KUKA KRL program: f1_Kuka_APT201T03S01.SRC

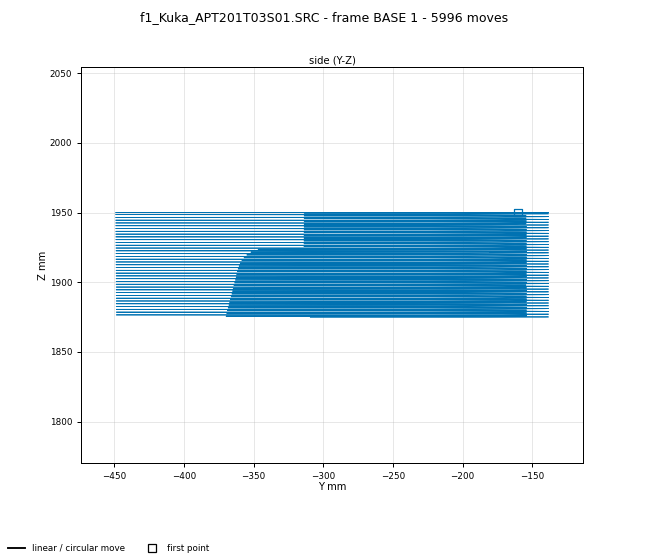
[picture p0: tool path of f1_Kuka_APT201T03S01.SRC in frame BASE 1, 5996 of 5998 moves have a stored position in this frame; points joined in program order, loops and branches not executed]
&ACCESS RVP
&REL 2
&PARAM TEMPLATE = C:\KRC\Roboter\Template\vorgabe
&PARAM EDITMASK = *
DEF f1_Kuka_APT201T03S01()


;FOLD INI;%{PE}%V3.2.0,%MKUKATPBASIS,%CINIT,%VCOMMON,%P
  ;FOLD BAS INI;%{E}%V3.2.0,%MKUKATPBASIS,%CINIT,%VINIT,%P
    GLOBAL INTERRUPT DECL 3 WHEN $STOPMESS==TRUE DO IR_STOPM ( )
    INTERRUPT ON 3
    BAS (#INITMOV,0 )
  ;ENDFOLD (BAS INI)
  ;FOLD USER INI;%{E}%V3.2.0,%MKUKATPUSER,%CINIT,%VINIT,%P
    ;Make your modifications here
  ;ENDFOLD (USER INI)
;ENDFOLD (INI)



;*** Make Initial Position Move
;FOLD PTP PPI1  Vel= 100 % PDAT1 Tool[0] Base[0];%{PE}%R 5.2.22,%MKUKATPBASIS,%CMOVE,%VPTP,%P 1:PTP, 2:PPI1, 3:, 5:100, 7:PDAT1
  $BWDSTART = FALSE
  PDAT_ACT = PPDAT1
  FDAT_ACT = FPPI1
  BAS(#PTP_PARAMS,100)
  PTP XPPI1
;ENDFOLD


;*** Auto Load the Correct TOOL and OFFSET
  ToolChange(3,1)


;*** Make Initial Position Move
;FOLD PTP PPI1  Vel= 100 % PDAT1 Tool[0] Base[0];%{PE}%R 5.2.22,%MKUKATPBASIS,%CMOVE,%VPTP,%P 1:PTP, 2:PPI1, 3:, 5:100, 7:PDAT1
  $BWDSTART = FALSE
  PDAT_ACT = PPDAT1
  FDAT_ACT = FPPI1
  BAS(#PTP_PARAMS,100)
  PTP XPPI1
;ENDFOLD

;*** Auto Load The Correct TOOL Data
  $tool=tool_data[3]

;*** Auto Load The Correct BASE Data
  $base=base_data[1]

  $ADVANCE = 5

SetRPM(6000)

MMPM(30000.0)
LIN {X 0.000,Y -160.097,Z 1950.000,A 0.000,B 0.000,C 90.000,E1 360.000} C_DIS
MMPM(15000.0)
LIN {X 0.000,Y -155.097,Z 1950.000,A 0.000,B 0.000,C 90.000,E1 360.000} C_DIS
MMPM(30000.0)
LIN {X -0.008,Y -154.165,Z 1950.000,A 0.000,B 0.000,C 90.000,E1 352.356} C_DIS
LIN {X -0.016,Y -155.912,Z 1950.000,A 0.000,B 0.000,C 90.000,E1 344.283} C_DIS
LIN {X 0.049,Y -158.612,Z 1950.000,A 0.000,B 0.000,C 90.000,E1 338.901} C_DIS
LIN {X 0.065,Y -162.189,Z 1950.000,A 0.000,B 0.000,C 90.000,E1 334.460} C_DIS
LIN {X -0.028,Y -166.034,Z 1950.000,A 0.000,B 0.000,C 90.000,E1 330.973} C_DIS
LIN {X 0.069,Y -170.880,Z 1950.000,A 0.000,B 0.000,C 90.000,E1 327.454} C_DIS
LIN {X -0.020,Y -175.155,Z 1950.000,A 0.000,B 0.000,C 90.000,E1 324.895} C_DIS
LIN {X -0.079,Y -180.105,Z 1950.000,A 0.000,B 0.000,C 90.000,E1 322.351} C_DIS
LIN {X 0.029,Y -185.957,Z 1950.000,A 0.000,B 0.000,C 90.000,E1 319.784} C_DIS
LIN {X -0.007,Y -191.568,Z 1950.000,A 0.000,B 0.000,C 90.000,E1 317.715} C_DIS
LIN {X 0.028,Y -199.262,Z 1950.000,A 0.000,B 0.000,C 90.000,E1 315.243} C_DIS
LIN {X -0.070,Y -207.846,Z 1950.000,A 0.000,B 0.000,C 90.000,E1 312.852} C_DIS
LIN {X -0.093,Y -218.894,Z 1950.000,A 0.000,B 0.000,C 90.000,E1 310.092} C_DIS
LIN {X -0.030,Y -232.809,Z 1950.000,A 0.000,B 0.000,C 90.000,E1 306.996} C_DIS
LIN {X 0.030,Y -247.857,Z 1950.000,A 0.000,B 0.000,C 90.000,E1 303.992} C_DIS
LIN {X 0.078,Y -259.781,Z 1950.000,A 0.000,B 0.000,C 90.000,E1 301.799} C_DIS
LIN {X 0.080,Y -271.838,Z 1950.000,A 0.000,B 0.000,C 90.000,E1 299.667} C_DIS
LIN {X -0.149,Y -281.753,Z 1950.000,A 0.000,B 0.000,C 90.000,E1 297.975} C_DIS
LIN {X 0.022,Y -291.348,Z 1950.000,A 0.000,B 0.000,C 90.000,E1 296.232} C_DIS
LIN {X 0.102,Y -296.741,Z 1950.000,A 0.000,B 0.000,C 90.000,E1 295.207} C_DIS
LIN {X 0.101,Y -301.534,Z 1950.000,A 0.000,B 0.000,C 90.000,E1 294.207} C_DIS
LIN {X -0.014,Y -304.343,Z 1950.000,A 0.000,B 0.000,C 90.000,E1 293.567} C_DIS
LIN {X 0.047,Y -306.751,Z 1950.000,A 0.000,B 0.000,C 90.000,E1 292.898} C_DIS
LIN {X -0.041,Y -308.757,Z 1950.000,A 0.000,B 0.000,C 90.000,E1 292.259} C_DIS
LIN {X 0.048,Y -310.413,Z 1950.000,A 0.000,B 0.000,C 90.000,E1 291.589} C_DIS
LIN {X 0.151,Y -311.750,Z 1950.000,A 0.000,B 0.000,C 90.000,E1 290.918} C_DIS
LIN {X -0.026,Y -312.741,Z 1950.000,A 0.000,B 0.000,C 90.000,E1 290.301} C_DIS
LIN {X 0.097,Y -313.399,Z 1950.000,A 0.000,B 0.000,C 90.000,E1 289.631} C_DIS
LIN {X -0.070,Y -313.739,Z 1950.000,A 0.000,B 0.000,C 90.000,E1 289.014} C_DIS
LIN {X -0.038,Y -313.728,Z 1950.000,A 0.000,B 0.000,C 90.000,E1 288.362} C_DIS
LIN {X 0.095,Y -313.339,Z 1950.000,A 0.000,B 0.000,C 90.000,E1 287.692} C_DIS
LIN {X 0.134,Y -312.501,Z 1950.000,A 0.000,B 0.000,C 90.000,E1 287.040} C_DIS
LIN {X -0.127,Y -311.193,Z 1950.000,A 0.000,B 0.000,C 90.000,E1 286.441} C_DIS
LIN {X -0.093,Y -309.374,Z 1950.000,A 0.000,B 0.000,C 90.000,E1 285.788} C_DIS
LIN {X -0.067,Y -306.893,Z 1950.000,A 0.000,B 0.000,C 90.000,E1 285.134} C_DIS
LIN {X -0.058,Y -303.660,Z 1950.000,A 0.000,B 0.000,C 90.000,E1 284.481} C_DIS
LIN {X -0.103,Y -295.919,Z 1950.000,A 0.000,B 0.000,C 90.000,E1 283.175} C_DIS
LIN {X -0.023,Y -290.732,Z 1950.000,A 0.000,B 0.000,C 90.000,E1 282.187} C_DIS
LIN {X -0.115,Y -286.366,Z 1950.000,A 0.000,B 0.000,C 90.000,E1 281.535} C_DIS
LIN {X -0.010,Y -281.038,Z 1950.000,A 0.000,B 0.000,C 90.000,E1 280.838} C_DIS
LIN {X -0.011,Y -274.872,Z 1950.000,A 0.000,B 0.000,C 90.000,E1 280.197} C_DIS
LIN {X 0.056,Y -268.439,Z 1950.000,A 0.000,B 0.000,C 90.000,E1 279.613} C_DIS
LIN {X 0.112,Y -261.807,Z 1950.000,A 0.000,B 0.000,C 90.000,E1 279.095} C_DIS
LIN {X -0.044,Y -255.112,Z 1950.000,A 0.000,B 0.000,C 90.000,E1 278.681} C_DIS
LIN {X 0.015,Y -248.167,Z 1950.000,A 0.000,B 0.000,C 90.000,E1 278.276} C_DIS
LIN {X 0.073,Y -240.768,Z 1950.000,A 0.000,B 0.000,C 90.000,E1 277.936} C_DIS
LIN {X -0.029,Y -232.686,Z 1950.000,A 0.000,B 0.000,C 90.000,E1 277.701} C_DIS
LIN {X -0.115,Y -222.350,Z 1950.000,A 0.000,B 0.000,C 90.000,E1 277.530} C_DIS
LIN {X -0.092,Y -214.660,Z 1950.000,A 0.000,B 0.000,C 90.000,E1 277.466} C_DIS
LIN {X 0.070,Y -180.206,Z 1950.000,A 0.000,B 0.000,C 90.000,E1 277.409} C_DIS
LIN {X 0.037,Y -181.028,Z 1950.000,A 0.000,B 0.000,C 90.000,E1 275.391} C_DIS
LIN {X 0.012,Y -181.579,Z 1950.000,A 0.000,B 0.000,C 90.000,E1 270.344} C_DIS
LIN {X -0.013,Y -180.904,Z 1950.000,A 0.000,B 0.000,C 90.000,E1 265.298} C_DIS
LIN {X -0.063,Y -180.241,Z 1950.000,A 0.000,B 0.000,C 90.000,E1 263.628} C_DIS
LIN {X -0.044,Y -178.728,Z 1950.000,A 0.000,B 0.000,C 90.000,E1 259.398} C_DIS
LIN {X 0.024,Y -175.777,Z 1950.000,A 0.000,B 0.000,C 90.000,E1 254.283} C_DIS
LIN {X 0.011,Y -171.961,Z 1950.000,A 0.000,B 0.000,C 90.000,E1 249.156} C_DIS
LIN {X 0.048,Y -171.355,Z 1950.000,A 0.000,B 0.000,C 90.000,E1 248.284} C_DIS
LIN {X 0.026,Y -167.605,Z 1950.000,A 0.000,B 0.000,C 90.000,E1 243.973} C_DIS
LIN {X 0.039,Y -166.250,Z 1950.000,A 0.000,B 0.000,C 90.000,E1 242.231} C_DIS
LIN {X 0.026,Y -163.005,Z 1950.000,A 0.000,B 0.000,C 90.000,E1 238.742} C_DIS
LIN {X 0.073,Y -160.927,Z 1950.000,A 0.000,B 0.000,C 90.000,E1 236.087} C_DIS
LIN {X 0.050,Y -157.689,Z 1950.000,A 0.000,B 0.000,C 90.000,E1 232.557} C_DIS
LIN {X -0.012,Y -155.727,Z 1950.000,A 0.000,B 0.000,C 90.000,E1 229.908} C_DIS
LIN {X 0.042,Y -151.987,Z 1950.000,A 0.000,B 0.000,C 90.000,E1 225.405} C_DIS
LIN {X 0.058,Y -150.231,Z 1950.000,A 0.000,B 0.000,C 90.000,E1 222.690} C_DIS
LIN {X -0.019,Y -146.992,Z 1950.000,A 0.000,B 0.000,C 90.000,E1 218.177} C_DIS
LIN {X -0.029,Y -145.577,Z 1950.000,A 0.000,B 0.000,C 90.000,E1 215.438} C_DIS
LIN {X -0.035,Y -142.967,Z 1950.000,A 0.000,B 0.000,C 90.000,E1 210.846} C_DIS
LIN {X 0.019,Y -141.593,Z 1950.000,A 0.000,B 0.000,C 90.000,E1 207.129} C_DIS
LIN {X 0.065,Y -139.421,Z 1950.000,A 0.000,B 0.000,C 90.000,E1 200.610} C_DIS
LIN {X -0.014,Y -139.148,Z 1950.000,A 0.000,B 0.000,C 90.000,E1 198.779} C_DIS
LIN {X 0.008,Y -138.346,Z 1950.000,A 0.000,B 0.000,C 90.000,E1 190.366} C_DIS
LIN {X -0.006,Y -139.487,Z 1950.000,A 0.000,B 0.000,C 90.000,E1 181.031} C_DIS
LIN {X -0.066,Y -141.091,Z 1950.000,A 0.000,B 0.000,C 90.000,E1 175.469} C_DIS
LIN {X 0.028,Y -142.469,Z 1950.000,A 0.000,B 0.000,C 90.000,E1 172.648} C_DIS
LIN {X -0.024,Y -144.713,Z 1950.000,A 0.000,B 0.000,C 90.000,E1 168.049} C_DIS
LIN {X 0.069,Y -147.314,Z 1950.000,A 0.000,B 0.000,C 90.000,E1 164.338} C_DIS
LIN {X -0.058,Y -150.634,Z 1950.000,A 0.000,B 0.000,C 90.000,E1 159.826} C_DIS
LIN {X 0.018,Y -154.111,Z 1950.000,A 0.000,B 0.000,C 90.000,E1 156.177} C_DIS
LIN {X -0.058,Y -157.536,Z 1950.000,A 0.000,B 0.000,C 90.000,E1 152.615} C_DIS
LIN {X 0.107,Y -161.773,Z 1950.000,A 0.000,B 0.000,C 90.000,E1 148.997} C_DIS
LIN {X -0.010,Y -165.966,Z 1950.000,A 0.000,B 0.000,C 90.000,E1 145.515} C_DIS
LIN {X -0.013,Y -170.959,Z 1950.000,A 0.000,B 0.000,C 90.000,E1 142.029} C_DIS
LIN {X 0.038,Y -175.828,Z 1950.000,A 0.000,B 0.000,C 90.000,E1 138.566} C_DIS
LIN {X 0.033,Y -181.435,Z 1950.000,A 0.000,B 0.000,C 90.000,E1 135.162} C_DIS
LIN {X -0.093,Y -186.940,Z 1950.000,A 0.000,B 0.000,C 90.000,E1 131.838} C_DIS
LIN {X -0.094,Y -190.052,Z 1950.000,A 0.000,B 0.000,C 90.000,E1 130.172} C_DIS
LIN {X -0.079,Y -195.827,Z 1950.000,A 0.000,B 0.000,C 90.000,E1 126.870} C_DIS
LIN {X -0.012,Y -200.659,Z 1950.000,A 0.000,B 0.000,C 90.000,E1 124.405} C_DIS
LIN {X 0.005,Y -206.543,Z 1950.000,A 0.000,B 0.000,C 90.000,E1 121.180} C_DIS
LIN {X -0.008,Y -209.835,Z 1950.000,A 0.000,B 0.000,C 90.000,E1 119.589} C_DIS
LIN {X -0.083,Y -217.193,Z 1950.000,A 0.000,B 0.000,C 90.000,E1 115.668} C_DIS
LIN {X 0.070,Y -218.819,Z 1950.000,A 0.000,B 0.000,C 90.000,E1 114.847} C_DIS
LIN {X 0.093,Y -224.206,Z 1950.000,A 0.000,B 0.000,C 90.000,E1 111.770} C_DIS
LIN {X 0.086,Y -283.482,Z 1950.000,A 0.000,B 0.000,C 90.000,E1 111.770} C_DIS
LIN {X -0.008,Y -285.142,Z 1950.000,A 0.000,B 0.000,C 90.000,E1 111.770} C_DIS
LIN {X -0.069,Y -288.414,Z 1950.000,A 0.000,B 0.000,C 90.000,E1 111.663} C_DIS
LIN {X 0.069,Y -291.624,Z 1950.000,A 0.000,B 0.000,C 90.000,E1 111.408} C_DIS
LIN {X 0.113,Y -295.303,Z 1950.000,A 0.000,B 0.000,C 90.000,E1 110.972} C_DIS
LIN {X 0.154,Y -300.812,Z 1950.000,A 0.000,B 0.000,C 90.000,E1 109.993} C_DIS
LIN {X 0.157,Y -314.505,Z 1950.000,A 0.000,B 0.000,C 90.000,E1 107.692} C_DIS
LIN {X -0.024,Y -329.600,Z 1950.000,A 0.000,B 0.000,C 90.000,E1 105.481} C_DIS
LIN {X 0.050,Y -343.764,Z 1950.000,A 0.000,B 0.000,C 90.000,E1 103.592} C_DIS
LIN {X 0.020,Y -359.097,Z 1950.000,A 0.000,B 0.000,C 90.000,E1 101.771} C_DIS
LIN {X 0.045,Y -377.683,Z 1950.000,A 0.000,B 0.000,C 90.000,E1 99.792} C_DIS
LIN {X 0.102,Y -396.651,Z 1950.000,A 0.000,B 0.000,C 90.000,E1 97.992} C_DIS
LIN {X 0.049,Y -418.788,Z 1950.000,A 0.000,B 0.000,C 90.000,E1 96.144} C_DIS
LIN {X 0.229,Y -438.507,Z 1950.000,A 0.000,B 0.000,C 90.000,E1 94.645} C_DIS
LIN {X -0.197,Y -442.974,Z 1950.000,A 0.000,B 0.000,C 90.000,E1 94.302} C_DIS
LIN {X 0.177,Y -446.090,Z 1950.000,A 0.000,B 0.000,C 90.000,E1 93.784} C_DIS
LIN {X -0.091,Y -447.256,Z 1950.000,A 0.000,B 0.000,C 90.000,E1 93.555} C_DIS
LIN {X 0.089,Y -448.110,Z 1950.000,A 0.000,B 0.000,C 90.000,E1 93.269} C_DIS
LIN {X 0.052,Y -449.023,Z 1950.000,A 0.000,B 0.000,C 90.000,E1 92.751} C_DIS
LIN {X -0.002,Y -448.993,Z 1950.000,A 0.000,B 0.000,C 90.000,E1 92.236} C_DIS
LIN {X -0.035,Y -448.019,Z 1950.000,A 0.000,B 0.000,C 90.000,E1 91.718} C_DIS
LIN {X -0.083,Y -445.945,Z 1950.000,A 0.000,B 0.000,C 90.000,E1 91.203} C_DIS
LIN {X -0.029,Y -437.820,Z 1950.000,A 0.000,B 0.000,C 90.000,E1 89.885} C_DIS
LIN {X 0.048,Y -427.895,Z 1950.000,A 0.000,B 0.000,C 90.000,E1 88.282} C_DIS
LIN {X 0.086,Y -416.100,Z 1950.000,A 0.000,B 0.000,C 90.000,E1 86.388} C_DIS
LIN {X -0.083,Y -404.293,Z 1950.000,A 0.000,B 0.000,C 90.000,E1 84.489} C_DIS
LIN {X -0.038,Y -392.326,Z 1950.000,A 0.000,B 0.000,C 90.000,E1 82.527} C_DIS
LIN {X 0.182,Y -380.404,Z 1950.000,A 0.000,B 0.000,C 90.000,E1 80.500} C_DIS
LIN {X -0.157,Y -368.656,Z 1950.000,A 0.000,B 0.000,C 90.000,E1 78.522} C_DIS
LIN {X 0.068,Y -352.618,Z 1950.000,A 0.000,B 0.000,C 90.000,E1 75.519} C_DIS
LIN {X 0.080,Y -338.999,Z 1950.000,A 0.000,B 0.000,C 90.000,E1 72.779} C_DIS
LIN {X -0.045,Y -327.232,Z 1950.000,A 0.000,B 0.000,C 90.000,E1 70.315} C_DIS
LIN {X -0.186,Y -314.366,Z 1950.000,A 0.000,B 0.000,C 90.000,E1 67.486} C_DIS
LIN {X 0.078,Y -303.504,Z 1950.000,A 0.000,B 0.000,C 90.000,E1 64.845} C_DIS
LIN {X -0.079,Y -291.384,Z 1950.000,A 0.000,B 0.000,C 90.000,E1 61.897} C_DIS
LIN {X -0.056,Y -283.397,Z 1950.000,A 0.000,B 0.000,C 90.000,E1 59.871} C_DIS
LIN {X 0.046,Y -273.868,Z 1950.000,A 0.000,B 0.000,C 90.000,E1 57.454} C_DIS
LIN {X -0.062,Y -265.672,Z 1950.000,A 0.000,B 0.000,C 90.000,E1 55.388} C_DIS
LIN {X -0.085,Y -254.640,Z 1950.000,A 0.000,B 0.000,C 90.000,E1 52.557} C_DIS
LIN {X 0.066,Y -245.071,Z 1950.000,A 0.000,B 0.000,C 90.000,E1 49.989} C_DIS
LIN {X -0.069,Y -234.340,Z 1950.000,A 0.000,B 0.000,C 90.000,E1 47.067} C_DIS
LIN {X -0.079,Y -225.290,Z 1950.000,A 0.000,B 0.000,C 90.000,E1 44.433} C_DIS
LIN {X 0.102,Y -215.369,Z 1950.000,A 0.000,B 0.000,C 90.000,E1 41.310} C_DIS
LIN {X 0.073,Y -206.134,Z 1950.000,A 0.000,B 0.000,C 90.000,E1 38.177} C_DIS
LIN {X -0.084,Y -197.783,Z 1950.000,A 0.000,B 0.000,C 90.000,E1 35.025} C_DIS
LIN {X -0.008,Y -190.163,Z 1950.000,A 0.000,B 0.000,C 90.000,E1 31.750} C_DIS
LIN {X 0.010,Y -183.313,Z 1950.000,A 0.000,B 0.000,C 90.000,E1 28.437} C_DIS
LIN {X 0.004,Y -177.164,Z 1950.000,A 0.000,B 0.000,C 90.000,E1 25.079} C_DIS
LIN {X 0.033,Y -171.845,Z 1950.000,A 0.000,B 0.000,C 90.000,E1 21.663} C_DIS
LIN {X -0.029,Y -167.319,Z 1950.000,A 0.000,B 0.000,C 90.000,E1 18.236} C_DIS
LIN {X 0.069,Y -163.659,Z 1950.000,A 0.000,B 0.000,C 90.000,E1 14.717} C_DIS
LIN {X -0.062,Y -159.917,Z 1950.000,A 0.000,B 0.000,C 90.000,E1 10.366} C_DIS
LIN {X -0.001,Y -157.330,Z 1950.000,A 0.000,B 0.000,C 90.000,E1 5.910} C_DIS
LIN {X -0.028,Y -154.972,Z 1949.997,A 0.000,B 0.000,C 90.000,E1 359.542} C_DIS
LIN {X 0.061,Y -154.207,Z 1949.953,A 0.000,B 0.000,C 90.000,E1 351.432} C_DIS
LIN {X -0.016,Y -155.911,Z 1949.913,A 0.000,B 0.000,C 90.000,E1 344.283} C_DIS
LIN {X 0.049,Y -158.611,Z 1949.883,A 0.000,B 0.000,C 90.000,E1 338.901} C_DIS
LIN {X 0.065,Y -162.188,Z 1949.858,A 0.000,B 0.000,C 90.000,E1 334.460} C_DIS
LIN {X -0.028,Y -166.034,Z 1949.839,A 0.000,B 0.000,C 90.000,E1 330.973} C_DIS
LIN {X 0.069,Y -170.880,Z 1949.819,A 0.000,B 0.000,C 90.000,E1 327.454} C_DIS
LIN {X -0.019,Y -175.156,Z 1949.805,A 0.000,B 0.000,C 90.000,E1 324.895} C_DIS
LIN {X -0.078,Y -180.105,Z 1949.791,A 0.000,B 0.000,C 90.000,E1 322.351} C_DIS
LIN {X 0.029,Y -185.958,Z 1949.777,A 0.000,B 0.000,C 90.000,E1 319.784} C_DIS
LIN {X -0.007,Y -191.569,Z 1949.765,A 0.000,B 0.000,C 90.000,E1 317.715} C_DIS
LIN {X 0.028,Y -199.262,Z 1949.751,A 0.000,B 0.000,C 90.000,E1 315.243} C_DIS
LIN {X -0.071,Y -207.847,Z 1949.738,A 0.000,B 0.000,C 90.000,E1 312.852} C_DIS
LIN {X -0.092,Y -218.894,Z 1949.723,A 0.000,B 0.000,C 90.000,E1 310.092} C_DIS
LIN {X -0.029,Y -232.810,Z 1949.705,A 0.000,B 0.000,C 90.000,E1 306.996} C_DIS
LIN {X 0.030,Y -247.859,Z 1949.689,A 0.000,B 0.000,C 90.000,E1 303.992} C_DIS
LIN {X 0.078,Y -259.783,Z 1949.677,A 0.000,B 0.000,C 90.000,E1 301.799} C_DIS
LIN {X 0.081,Y -271.839,Z 1949.665,A 0.000,B 0.000,C 90.000,E1 299.667} C_DIS
LIN {X -0.148,Y -281.754,Z 1949.655,A 0.000,B 0.000,C 90.000,E1 297.975} C_DIS
LIN {X 0.022,Y -291.349,Z 1949.646,A 0.000,B 0.000,C 90.000,E1 296.232} C_DIS
LIN {X 0.102,Y -296.743,Z 1949.640,A 0.000,B 0.000,C 90.000,E1 295.207} C_DIS
LIN {X 0.102,Y -301.537,Z 1949.635,A 0.000,B 0.000,C 90.000,E1 294.207} C_DIS
LIN {X -0.014,Y -304.344,Z 1949.631,A 0.000,B 0.000,C 90.000,E1 293.567} C_DIS
LIN {X 0.047,Y -306.753,Z 1949.627,A 0.000,B 0.000,C 90.000,E1 292.898} C_DIS
LIN {X -0.040,Y -308.760,Z 1949.624,A 0.000,B 0.000,C 90.000,E1 292.259} C_DIS
LIN {X 0.048,Y -310.415,Z 1949.620,A 0.000,B 0.000,C 90.000,E1 291.589} C_DIS
LIN {X 0.152,Y -311.752,Z 1949.616,A 0.000,B 0.000,C 90.000,E1 290.918} C_DIS
LIN {X -0.026,Y -312.743,Z 1949.613,A 0.000,B 0.000,C 90.000,E1 290.301} C_DIS
LIN {X 0.097,Y -313.402,Z 1949.609,A 0.000,B 0.000,C 90.000,E1 289.631} C_DIS
LIN {X -0.070,Y -313.742,Z 1949.606,A 0.000,B 0.000,C 90.000,E1 289.014} C_DIS
LIN {X -0.038,Y -313.731,Z 1949.602,A 0.000,B 0.000,C 90.000,E1 288.362} C_DIS
LIN {X 0.096,Y -313.342,Z 1949.598,A 0.000,B 0.000,C 90.000,E1 287.692} C_DIS
LIN {X 0.134,Y -312.505,Z 1949.595,A 0.000,B 0.000,C 90.000,E1 287.040} C_DIS
LIN {X -0.127,Y -311.196,Z 1949.591,A 0.000,B 0.000,C 90.000,E1 286.441} C_DIS
LIN {X -0.092,Y -309.377,Z 1949.588,A 0.000,B 0.000,C 90.000,E1 285.788} C_DIS
LIN {X -0.065,Y -306.896,Z 1949.584,A 0.000,B 0.000,C 90.000,E1 285.134} C_DIS
LIN {X -0.057,Y -303.664,Z 1949.580,A 0.000,B 0.000,C 90.000,E1 284.481} C_DIS
LIN {X 0.025,Y -297.714,Z 1949.575,A 0.000,B 0.000,C 90.000,E1 283.480} C_DIS
LIN {X -0.023,Y -290.734,Z 1949.568,A 0.000,B 0.000,C 90.000,E1 282.187} C_DIS
LIN {X -0.116,Y -286.368,Z 1949.564,A 0.000,B 0.000,C 90.000,E1 281.535} C_DIS
LIN {X -0.009,Y -281.040,Z 1949.560,A 0.000,B 0.000,C 90.000,E1 280.838} C_DIS
LIN {X -0.011,Y -274.872,Z 1949.557,A 0.000,B 0.000,C 90.000,E1 280.197} C_DIS
LIN {X 0.056,Y -268.439,Z 1949.553,A 0.000,B 0.000,C 90.000,E1 279.613} C_DIS
LIN {X 0.112,Y -261.806,Z 1949.551,A 0.000,B 0.000,C 90.000,E1 279.095} C_DIS
LIN {X -0.043,Y -255.109,Z 1949.548,A 0.000,B 0.000,C 90.000,E1 278.681} C_DIS
LIN {X 0.015,Y -248.163,Z 1949.546,A 0.000,B 0.000,C 90.000,E1 278.276} C_DIS
LIN {X 0.071,Y -240.761,Z 1949.544,A 0.000,B 0.000,C 90.000,E1 277.936} C_DIS
LIN {X -0.029,Y -232.680,Z 1949.543,A 0.000,B 0.000,C 90.000,E1 277.701} C_DIS
LIN {X -0.114,Y -222.330,Z 1949.542,A 0.000,B 0.000,C 90.000,E1 277.530} C_DIS
LIN {X -0.091,Y -214.438,Z 1949.541,A 0.000,B 0.000,C 90.000,E1 277.466} C_DIS
LIN {X 0.070,Y -180.205,Z 1949.541,A 0.000,B 0.000,C 90.000,E1 277.409} C_DIS
LIN {X 0.037,Y -181.028,Z 1949.530,A 0.000,B 0.000,C 90.000,E1 275.391} C_DIS
LIN {X 0.012,Y -181.579,Z 1949.502,A 0.000,B 0.000,C 90.000,E1 270.344} C_DIS
LIN {X -0.012,Y -180.904,Z 1949.474,A 0.000,B 0.000,C 90.000,E1 265.298} C_DIS
LIN {X -0.062,Y -180.241,Z 1949.464,A 0.000,B 0.000,C 90.000,E1 263.628} C_DIS
LIN {X -0.043,Y -178.728,Z 1949.441,A 0.000,B 0.000,C 90.000,E1 259.398} C_DIS
LIN {X 0.024,Y -175.777,Z 1949.413,A 0.000,B 0.000,C 90.000,E1 254.283} C_DIS
LIN {X 0.012,Y -171.960,Z 1949.384,A 0.000,B 0.000,C 90.000,E1 249.156} C_DIS
LIN {X 0.048,Y -171.355,Z 1949.379,A 0.000,B 0.000,C 90.000,E1 248.284} C_DIS
LIN {X 0.027,Y -167.605,Z 1949.355,A 0.000,B 0.000,C 90.000,E1 243.973} C_DIS
LIN {X 0.039,Y -166.250,Z 1949.346,A 0.000,B 0.000,C 90.000,E1 242.231} C_DIS
LIN {X 0.027,Y -163.006,Z 1949.326,A 0.000,B 0.000,C 90.000,E1 238.742} C_DIS
LIN {X 0.073,Y -160.927,Z 1949.312,A 0.000,B 0.000,C 90.000,E1 236.087} C_DIS
LIN {X 0.050,Y -157.689,Z 1949.292,A 0.000,B 0.000,C 90.000,E1 232.557} C_DIS
LIN {X -0.012,Y -155.727,Z 1949.277,A 0.000,B 0.000,C 90.000,E1 229.908} C_DIS
LIN {X 0.042,Y -151.987,Z 1949.252,A 0.000,B 0.000,C 90.000,E1 225.405} C_DIS
LIN {X 0.058,Y -150.231,Z 1949.237,A 0.000,B 0.000,C 90.000,E1 222.690} C_DIS
LIN {X -0.019,Y -146.992,Z 1949.212,A 0.000,B 0.000,C 90.000,E1 218.177} C_DIS
LIN {X -0.028,Y -145.578,Z 1949.197,A 0.000,B 0.000,C 90.000,E1 215.438} C_DIS
LIN {X -0.035,Y -142.967,Z 1949.171,A 0.000,B 0.000,C 90.000,E1 210.846} C_DIS
LIN {X 0.020,Y -141.594,Z 1949.151,A 0.000,B 0.000,C 90.000,E1 207.129} C_DIS
LIN {X 0.066,Y -139.421,Z 1949.115,A 0.000,B 0.000,C 90.000,E1 200.610} C_DIS
LIN {X -0.014,Y -139.148,Z 1949.104,A 0.000,B 0.000,C 90.000,E1 198.779} C_DIS
LIN {X 0.009,Y -138.346,Z 1949.058,A 0.000,B 0.000,C 90.000,E1 190.366} C_DIS
LIN {X -0.006,Y -139.487,Z 1949.006,A 0.000,B 0.000,C 90.000,E1 181.031} C_DIS
LIN {X -0.065,Y -141.090,Z 1948.975,A 0.000,B 0.000,C 90.000,E1 175.469} C_DIS
LIN {X 0.028,Y -142.468,Z 1948.959,A 0.000,B 0.000,C 90.000,E1 172.648} C_DIS
LIN {X -0.024,Y -144.713,Z 1948.934,A 0.000,B 0.000,C 90.000,E1 168.049} C_DIS
LIN {X 0.070,Y -147.314,Z 1948.913,A 0.000,B 0.000,C 90.000,E1 164.338} C_DIS
LIN {X -0.058,Y -150.634,Z 1948.888,A 0.000,B 0.000,C 90.000,E1 159.826} C_DIS
LIN {X 0.018,Y -154.111,Z 1948.868,A 0.000,B 0.000,C 90.000,E1 156.177} C_DIS
LIN {X -0.058,Y -157.536,Z 1948.848,A 0.000,B 0.000,C 90.000,E1 152.615} C_DIS
LIN {X 0.108,Y -161.772,Z 1948.828,A 0.000,B 0.000,C 90.000,E1 148.997} C_DIS
LIN {X -0.009,Y -165.965,Z 1948.808,A 0.000,B 0.000,C 90.000,E1 145.515} C_DIS
LIN {X -0.012,Y -170.959,Z 1948.789,A 0.000,B 0.000,C 90.000,E1 142.029} C_DIS
LIN {X 0.039,Y -175.827,Z 1948.770,A 0.000,B 0.000,C 90.000,E1 138.566} C_DIS
LIN {X 0.034,Y -181.435,Z 1948.751,A 0.000,B 0.000,C 90.000,E1 135.162} C_DIS
LIN {X -0.092,Y -186.939,Z 1948.732,A 0.000,B 0.000,C 90.000,E1 131.838} C_DIS
LIN {X -0.093,Y -190.052,Z 1948.723,A 0.000,B 0.000,C 90.000,E1 130.172} C_DIS
LIN {X -0.079,Y -195.827,Z 1948.705,A 0.000,B 0.000,C 90.000,E1 126.870} C_DIS
LIN {X -0.011,Y -200.658,Z 1948.691,A 0.000,B 0.000,C 90.000,E1 124.405} C_DIS
LIN {X 0.005,Y -206.543,Z 1948.673,A 0.000,B 0.000,C 90.000,E1 121.180} C_DIS
LIN {X -0.008,Y -209.834,Z 1948.664,A 0.000,B 0.000,C 90.000,E1 119.589} C_DIS
LIN {X -0.082,Y -217.192,Z 1948.642,A 0.000,B 0.000,C 90.000,E1 115.668} C_DIS
LIN {X 0.070,Y -218.819,Z 1948.638,A 0.000,B 0.000,C 90.000,E1 114.847} C_DIS
LIN {X 0.094,Y -224.205,Z 1948.621,A 0.000,B 0.000,C 90.000,E1 111.770} C_DIS
LIN {X 0.087,Y -283.684,Z 1948.621,A 0.000,B 0.000,C 90.000,E1 111.770} C_DIS
LIN {X -0.008,Y -285.184,Z 1948.621,A 0.000,B 0.000,C 90.000,E1 111.770} C_DIS
LIN {X -0.082,Y -288.479,Z 1948.620,A 0.000,B 0.000,C 90.000,E1 111.663} C_DIS
LIN {X 0.037,Y -291.700,Z 1948.619,A 0.000,B 0.000,C 90.000,E1 111.408} C_DIS
LIN {X 0.057,Y -295.379,Z 1948.617,A 0.000,B 0.000,C 90.000,E1 110.972} C_DIS
LIN {X -0.059,Y -302.779,Z 1948.609,A 0.000,B 0.000,C 90.000,E1 109.685} C_DIS
LIN {X -0.112,Y -316.669,Z 1948.597,A 0.000,B 0.000,C 90.000,E1 107.402} C_DIS
LIN {X 0.062,Y -331.994,Z 1948.584,A 0.000,B 0.000,C 90.000,E1 105.134} C_DIS
LIN {X -0.144,Y -346.365,Z 1948.574,A 0.000,B 0.000,C 90.000,E1 103.300} C_DIS
LIN {X -0.091,Y -361.864,Z 1948.564,A 0.000,B 0.000,C 90.000,E1 101.478} C_DIS
LIN {X 0.141,Y -380.481,Z 1948.553,A 0.000,B 0.000,C 90.000,E1 99.500} C_DIS
LIN {X -0.045,Y -399.543,Z 1948.543,A 0.000,B 0.000,C 90.000,E1 97.757} C_DIS
LIN {X 0.073,Y -421.735,Z 1948.533,A 0.000,B 0.000,C 90.000,E1 95.910} C_DIS
LIN {X 0.155,Y -438.642,Z 1948.526,A 0.000,B 0.000,C 90.000,E1 94.645} C_DIS
LIN {X 0.171,Y -443.048,Z 1948.524,A 0.000,B 0.000,C 90.000,E1 94.245} C_DIS
LIN {X 0.070,Y -446.151,Z 1948.521,A 0.000,B 0.000,C 90.000,E1 93.784} C_DIS
LIN {X -0.197,Y -447.298,Z 1948.520,A 0.000,B 0.000,C 90.000,E1 93.555} C_DIS
LIN {X -0.016,Y -448.137,Z 1948.518,A 0.000,B 0.000,C 90.000,E1 93.269} C_DIS
LIN {X -0.054,Y -449.023,Z 1948.515,A 0.000,B 0.000,C 90.000,E1 92.751} C_DIS
LIN {X -0.108,Y -448.969,Z 1948.512,A 0.000,B 0.000,C 90.000,E1 92.236} C_DIS
LIN {X -0.140,Y -447.968,Z 1948.509,A 0.000,B 0.000,C 90.000,E1 91.718} C_DIS
LIN {X -0.188,Y -445.858,Z 1948.507,A 0.000,B 0.000,C 90.000,E1 91.203} C_DIS
LIN {X 0.040,Y -436.074,Z 1948.498,A 0.000,B 0.000,C 90.000,E1 89.599} C_DIS
LIN {X 0.098,Y -426.119,Z 1948.489,A 0.000,B 0.000,C 90.000,E1 87.993} C_DIS
LIN {X 0.198,Y -412.640,Z 1948.477,A 0.000,B 0.000,C 90.000,E1 85.812} C_DIS
LIN {X -0.127,Y -402.486,Z 1948.468,A 0.000,B 0.000,C 90.000,E1 84.204} C_DIS
LIN {X -0.132,Y -390.500,Z 1948.457,A 0.000,B 0.000,C 90.000,E1 82.243} C_DIS
LIN {X 0.113,Y -378.618,Z 1948.446,A 0.000,B 0.000,C 90.000,E1 80.208} C_DIS
LIN {X 0.085,Y -365.258,Z 1948.433,A 0.000,B 0.000,C 90.000,E1 77.881} C_DIS
LIN {X -0.128,Y -347.919,Z 1948.415,A 0.000,B 0.000,C 90.000,E1 74.629} C_DIS
LIN {X -0.132,Y -334.473,Z 1948.399,A 0.000,B 0.000,C 90.000,E1 71.873} C_DIS
LIN {X 0.054,Y -322.786,Z 1948.385,A 0.000,B 0.000,C 90.000,E1 69.337} C_DIS
LIN {X -0.175,Y -308.805,Z 1948.367,A 0.000,B 0.000,C 90.000,E1 66.177} C_DIS
LIN {X -0.096,Y -300.700,Z 1948.357,A 0.000,B 0.000,C 90.000,E1 64.204} C_DIS
LIN {X 0.069,Y -288.652,Z 1948.340,A 0.000,B 0.000,C 90.000,E1 61.179} C_DIS
LIN {X 0.035,Y -280.597,Z 1948.329,A 0.000,B 0.000,C 90.000,E1 59.154} C_DIS
LIN {X -0.014,Y -271.049,Z 1948.315,A 0.000,B 0.000,C 90.000,E1 56.755} C_DIS
LIN {X 0.046,Y -262.799,Z 1948.304,A 0.000,B 0.000,C 90.000,E1 54.642} C_DIS
LIN {X -0.106,Y -251.813,Z 1948.288,A 0.000,B 0.000,C 90.000,E1 51.823} C_DIS
LIN {X -0.017,Y -242.245,Z 1948.274,A 0.000,B 0.000,C 90.000,E1 49.256} C_DIS
LIN {X -0.064,Y -231.651,Z 1948.257,A 0.000,B 0.000,C 90.000,E1 46.296} C_DIS
LIN {X -0.046,Y -221.401,Z 1948.240,A 0.000,B 0.000,C 90.000,E1 43.257} C_DIS
LIN {X 0.103,Y -210.572,Z 1948.221,A 0.000,B 0.000,C 90.000,E1 39.725} C_DIS
LIN {X -0.002,Y -201.783,Z 1948.203,A 0.000,B 0.000,C 90.000,E1 36.583} C_DIS
LIN {X -0.047,Y -193.820,Z 1948.185,A 0.000,B 0.000,C 90.000,E1 33.372} C_DIS
LIN {X -0.007,Y -186.580,Z 1948.167,A 0.000,B 0.000,C 90.000,E1 30.079} C_DIS
LIN {X -0.007,Y -180.107,Z 1948.149,A 0.000,B 0.000,C 90.000,E1 26.744} C_DIS
LIN {X 0.006,Y -175.712,Z 1948.135,A 0.000,B 0.000,C 90.000,E1 24.207} C_DIS
LIN {X 0.001,Y -170.592,Z 1948.115,A 0.000,B 0.000,C 90.000,E1 20.791} C_DIS
LIN {X 0.008,Y -166.304,Z 1948.096,A 0.000,B 0.000,C 90.000,E1 17.330} C_DIS
LIN {X 0.067,Y -162.018,Z 1948.072,A 0.000,B 0.000,C 90.000,E1 12.939} C_DIS
LIN {X -0.025,Y -159.285,Z 1948.052,A 0.000,B 0.000,C 90.000,E1 9.443} C_DIS
LIN {X -0.077,Y -156.526,Z 1948.023,A 0.000,B 0.000,C 90.000,E1 4.131} C_DIS
LIN {X -0.010,Y -154.445,Z 1947.982,A 0.000,B 0.000,C 90.000,E1 356.846} C_DIS
LIN {X 0.001,Y -155.589,Z 1947.918,A 0.000,B 0.000,C 90.000,E1 345.172} C_DIS
LIN {X -0.047,Y -158.036,Z 1947.888,A 0.000,B 0.000,C 90.000,E1 339.826} C_DIS
LIN {X 0.028,Y -161.378,Z 1947.863,A 0.000,B 0.000,C 90.000,E1 335.357} C_DIS
LIN {X -0.019,Y -164.979,Z 1947.844,A 0.000,B 0.000,C 90.000,E1 331.847} C_DIS
LIN {X 0.048,Y -169.590,Z 1947.824,A 0.000,B 0.000,C 90.000,E1 328.329} C_DIS
LIN {X -0.016,Y -173.665,Z 1947.810,A 0.000,B 0.000,C 90.000,E1 325.754} C_DIS
LIN {X 0.003,Y -178.369,Z 1947.795,A 0.000,B 0.000,C 90.000,E1 323.176} C_DIS
LIN {X -0.027,Y -183.919,Z 1947.781,A 0.000,B 0.000,C 90.000,E1 320.642} C_DIS
LIN {X 0.044,Y -189.229,Z 1947.770,A 0.000,B 0.000,C 90.000,E1 318.528} C_DIS
LIN {X 0.047,Y -196.615,Z 1947.756,A 0.000,B 0.000,C 90.000,E1 316.053} C_DIS
LIN {X 0.040,Y -204.887,Z 1947.742,A 0.000,B 0.000,C 90.000,E1 313.623} C_DIS
LIN {X -0.045,Y -215.645,Z 1947.727,A 0.000,B 0.000,C 90.000,E1 310.862} C_DIS
LIN {X 0.148,Y -227.444,Z 1947.712,A 0.000,B 0.000,C 90.000,E1 308.096} C_DIS
LIN {X 0.023,Y -242.095,Z 1947.695,A 0.000,B 0.000,C 90.000,E1 305.105} C_DIS
LIN {X -0.035,Y -255.800,Z 1947.681,A 0.000,B 0.000,C 90.000,E1 302.546} C_DIS
LIN {X 0.023,Y -267.810,Z 1947.669,A 0.000,B 0.000,C 90.000,E1 300.384} C_DIS
LIN {X 0.105,Y -277.832,Z 1947.659,A 0.000,B 0.000,C 90.000,E1 298.615} C_DIS
LIN {X -0.039,Y -287.574,Z 1947.650,A 0.000,B 0.000,C 90.000,E1 296.924} C_DIS
LIN {X 0.114,Y -295.003,Z 1947.642,A 0.000,B 0.000,C 90.000,E1 295.540} C_DIS
LIN {X -0.041,Y -300.028,Z 1947.636,A 0.000,B 0.000,C 90.000,E1 294.567} C_DIS
LIN {X -0.015,Y -303.010,Z 1947.633,A 0.000,B 0.000,C 90.000,E1 293.898} C_DIS
LIN {X 0.048,Y -306.765,Z 1947.627,A 0.000,B 0.000,C 90.000,E1 292.898} C_DIS
LIN {X -0.038,Y -308.772,Z 1947.624,A 0.000,B 0.000,C 90.000,E1 292.259} C_DIS
LIN {X 0.050,Y -310.430,Z 1947.620,A 0.000,B 0.000,C 90.000,E1 291.589} C_DIS
LIN {X 0.153,Y -311.768,Z 1947.616,A 0.000,B 0.000,C 90.000,E1 290.918} C_DIS
LIN {X -0.024,Y -312.760,Z 1947.613,A 0.000,B 0.000,C 90.000,E1 290.301} C_DIS
LIN {X 0.099,Y -313.415,Z 1947.609,A 0.000,B 0.000,C 90.000,E1 289.631} C_DIS
LIN {X -0.067,Y -313.757,Z 1947.606,A 0.000,B 0.000,C 90.000,E1 289.014} C_DIS
LIN {X -0.036,Y -313.745,Z 1947.602,A 0.000,B 0.000,C 90.000,E1 288.362} C_DIS
LIN {X 0.098,Y -313.357,Z 1947.598,A 0.000,B 0.000,C 90.000,E1 287.692} C_DIS
LIN {X 0.136,Y -312.523,Z 1947.595,A 0.000,B 0.000,C 90.000,E1 287.040} C_DIS
LIN {X -0.125,Y -311.211,Z 1947.591,A 0.000,B 0.000,C 90.000,E1 286.441} C_DIS
LIN {X -0.090,Y -309.392,Z 1947.588,A 0.000,B 0.000,C 90.000,E1 285.788} C_DIS
LIN {X -0.063,Y -306.916,Z 1947.584,A 0.000,B 0.000,C 90.000,E1 285.134} C_DIS
LIN {X -0.055,Y -303.682,Z 1947.580,A 0.000,B 0.000,C 90.000,E1 284.481} C_DIS
LIN {X 0.028,Y -297.730,Z 1947.575,A 0.000,B 0.000,C 90.000,E1 283.480} C_DIS
LIN {X -0.022,Y -290.745,Z 1947.568,A 0.000,B 0.000,C 90.000,E1 282.187} C_DIS
LIN {X -0.114,Y -286.375,Z 1947.564,A 0.000,B 0.000,C 90.000,E1 281.535} C_DIS
LIN {X -0.008,Y -281.049,Z 1947.560,A 0.000,B 0.000,C 90.000,E1 280.838} C_DIS
LIN {X -0.009,Y -274.872,Z 1947.557,A 0.000,B 0.000,C 90.000,E1 280.197} C_DIS
LIN {X 0.056,Y -268.438,Z 1947.553,A 0.000,B 0.000,C 90.000,E1 279.613} C_DIS
LIN {X 0.110,Y -261.800,Z 1947.551,A 0.000,B 0.000,C 90.000,E1 279.095} C_DIS
LIN {X -0.045,Y -255.094,Z 1947.548,A 0.000,B 0.000,C 90.000,E1 278.681} C_DIS
LIN {X 0.013,Y -248.148,Z 1947.546,A 0.000,B 0.000,C 90.000,E1 278.276} C_DIS
LIN {X 0.071,Y -240.731,Z 1947.544,A 0.000,B 0.000,C 90.000,E1 277.936} C_DIS
LIN {X -0.030,Y -232.649,Z 1947.543,A 0.000,B 0.000,C 90.000,E1 277.701} C_DIS
LIN {X -0.114,Y -222.243,Z 1947.542,A 0.000,B 0.000,C 90.000,E1 277.530} C_DIS
LIN {X -0.090,Y -213.337,Z 1947.541,A 0.000,B 0.000,C 90.000,E1 277.466} C_DIS
LIN {X 0.071,Y -180.205,Z 1947.541,A 0.000,B 0.000,C 90.000,E1 277.409} C_DIS
LIN {X 0.039,Y -181.029,Z 1947.530,A 0.000,B 0.000,C 90.000,E1 275.391} C_DIS
LIN {X 0.014,Y -181.579,Z 1947.502,A 0.000,B 0.000,C 90.000,E1 270.344} C_DIS
LIN {X -0.011,Y -180.904,Z 1947.474,A 0.000,B 0.000,C 90.000,E1 265.298} C_DIS
LIN {X -0.061,Y -180.242,Z 1947.464,A 0.000,B 0.000,C 90.000,E1 263.628} C_DIS
LIN {X -0.042,Y -178.729,Z 1947.441,A 0.000,B 0.000,C 90.000,E1 259.398} C_DIS
LIN {X 0.025,Y -175.776,Z 1947.413,A 0.000,B 0.000,C 90.000,E1 254.283} C_DIS
LIN {X 0.014,Y -171.961,Z 1947.384,A 0.000,B 0.000,C 90.000,E1 249.156} C_DIS
LIN {X 0.051,Y -171.355,Z 1947.379,A 0.000,B 0.000,C 90.000,E1 248.284} C_DIS
LIN {X 0.029,Y -167.605,Z 1947.355,A 0.000,B 0.000,C 90.000,E1 243.973} C_DIS
LIN {X 0.040,Y -166.250,Z 1947.346,A 0.000,B 0.000,C 90.000,E1 242.231} C_DIS
LIN {X 0.029,Y -163.006,Z 1947.326,A 0.000,B 0.000,C 90.000,E1 238.742} C_DIS
LIN {X 0.075,Y -160.928,Z 1947.312,A 0.000,B 0.000,C 90.000,E1 236.087} C_DIS
LIN {X 0.052,Y -157.689,Z 1947.292,A 0.000,B 0.000,C 90.000,E1 232.557} C_DIS
LIN {X -0.010,Y -155.728,Z 1947.277,A 0.000,B 0.000,C 90.000,E1 229.908} C_DIS
LIN {X 0.044,Y -151.987,Z 1947.252,A 0.000,B 0.000,C 90.000,E1 225.405} C_DIS
LIN {X 0.060,Y -150.232,Z 1947.237,A 0.000,B 0.000,C 90.000,E1 222.690} C_DIS
LIN {X -0.017,Y -146.993,Z 1947.212,A 0.000,B 0.000,C 90.000,E1 218.177} C_DIS
LIN {X -0.027,Y -145.578,Z 1947.197,A 0.000,B 0.000,C 90.000,E1 215.438} C_DIS
LIN {X -0.032,Y -142.967,Z 1947.171,A 0.000,B 0.000,C 90.000,E1 210.846} C_DIS
LIN {X 0.021,Y -141.594,Z 1947.151,A 0.000,B 0.000,C 90.000,E1 207.129} C_DIS
LIN {X 0.067,Y -139.421,Z 1947.115,A 0.000,B 0.000,C 90.000,E1 200.610} C_DIS
LIN {X -0.012,Y -139.147,Z 1947.104,A 0.000,B 0.000,C 90.000,E1 198.779} C_DIS
LIN {X 0.010,Y -138.346,Z 1947.058,A 0.000,B 0.000,C 90.000,E1 190.366} C_DIS
LIN {X -0.005,Y -139.487,Z 1947.006,A 0.000,B 0.000,C 90.000,E1 181.031} C_DIS
LIN {X -0.064,Y -141.090,Z 1946.975,A 0.000,B 0.000,C 90.000,E1 175.469} C_DIS
LIN {X 0.030,Y -142.468,Z 1946.959,A 0.000,B 0.000,C 90.000,E1 172.648} C_DIS
LIN {X -0.022,Y -144.713,Z 1946.934,A 0.000,B 0.000,C 90.000,E1 168.049} C_DIS
LIN {X -0.071,Y -147.314,Z 1946.913,A 0.000,B 0.000,C 90.000,E1 164.393} C_DIS
LIN {X -0.056,Y -150.634,Z 1946.888,A 0.000,B 0.000,C 90.000,E1 159.826} C_DIS
LIN {X 0.020,Y -154.111,Z 1946.868,A 0.000,B 0.000,C 90.000,E1 156.177} C_DIS
LIN {X -0.056,Y -157.535,Z 1946.848,A 0.000,B 0.000,C 90.000,E1 152.615} C_DIS
LIN {X 0.109,Y -161.772,Z 1946.828,A 0.000,B 0.000,C 90.000,E1 148.997} C_DIS
LIN {X -0.007,Y -165.964,Z 1946.808,A 0.000,B 0.000,C 90.000,E1 145.515} C_DIS
LIN {X -0.011,Y -170.958,Z 1946.789,A 0.000,B 0.000,C 90.000,E1 142.029} C_DIS
LIN {X 0.040,Y -175.827,Z 1946.770,A 0.000,B 0.000,C 90.000,E1 138.566} C_DIS
LIN {X 0.035,Y -181.433,Z 1946.751,A 0.000,B 0.000,C 90.000,E1 135.162} C_DIS
LIN {X -0.091,Y -186.939,Z 1946.732,A 0.000,B 0.000,C 90.000,E1 131.838} C_DIS
LIN {X -0.091,Y -190.051,Z 1946.723,A 0.000,B 0.000,C 90.000,E1 130.172} C_DIS
LIN {X -0.077,Y -195.826,Z 1946.705,A 0.000,B 0.000,C 90.000,E1 126.870} C_DIS
LIN {X -0.010,Y -200.657,Z 1946.691,A 0.000,B 0.000,C 90.000,E1 124.405} C_DIS
LIN {X 0.007,Y -206.542,Z 1946.673,A 0.000,B 0.000,C 90.000,E1 121.180} C_DIS
LIN {X -0.006,Y -209.834,Z 1946.664,A 0.000,B 0.000,C 90.000,E1 119.589} C_DIS
LIN {X -0.080,Y -217.192,Z 1946.642,A 0.000,B 0.000,C 90.000,E1 115.668} C_DIS
LIN {X 0.072,Y -218.818,Z 1946.638,A 0.000,B 0.000,C 90.000,E1 114.847} C_DIS
LIN {X 0.096,Y -224.204,Z 1946.621,A 0.000,B 0.000,C 90.000,E1 111.770} C_DIS
LIN {X 0.090,Y -283.852,Z 1946.621,A 0.000,B 0.000,C 90.000,E1 111.770} C_DIS
LIN {X -0.005,Y -285.231,Z 1946.621,A 0.000,B 0.000,C 90.000,E1 111.770} C_DIS
LIN {X -0.097,Y -288.551,Z 1946.620,A 0.000,B 0.000,C 90.000,E1 111.663} C_DIS
LIN {X 0.000,Y -291.787,Z 1946.619,A 0.000,B 0.000,C 90.000,E1 111.408} C_DIS
LIN {X -0.009,Y -295.466,Z 1946.616,A 0.000,B 0.000,C 90.000,E1 110.972} C_DIS
LIN {X -0.023,Y -308.674,Z 1946.604,A 0.000,B 0.000,C 90.000,E1 108.671} C_DIS
LIN {X 0.064,Y -323.178,Z 1946.591,A 0.000,B 0.000,C 90.000,E1 106.386} C_DIS
LIN {X 0.108,Y -336.785,Z 1946.581,A 0.000,B 0.000,C 90.000,E1 104.481} C_DIS
LIN {X -0.008,Y -351.570,Z 1946.570,A 0.000,B 0.000,C 90.000,E1 102.647} C_DIS
LIN {X -0.051,Y -369.927,Z 1946.559,A 0.000,B 0.000,C 90.000,E1 100.602} C_DIS
LIN {X -0.130,Y -388.765,Z 1946.548,A 0.000,B 0.000,C 90.000,E1 98.746} C_DIS
LIN {X 0.137,Y -407.950,Z 1946.539,A 0.000,B 0.000,C 90.000,E1 97.011} C_DIS
LIN {X -0.054,Y -430.301,Z 1946.529,A 0.000,B 0.000,C 90.000,E1 95.277} C_DIS
LIN {X 0.068,Y -438.800,Z 1946.526,A 0.000,B 0.000,C 90.000,E1 94.645} C_DIS
LIN {X 0.087,Y -443.133,Z 1946.524,A 0.000,B 0.000,C 90.000,E1 94.245} C_DIS
LIN {X -0.054,Y -446.221,Z 1946.521,A 0.000,B 0.000,C 90.000,E1 93.784} C_DIS
LIN {X -0.141,Y -448.166,Z 1946.518,A 0.000,B 0.000,C 90.000,E1 93.269} C_DIS
LIN {X -0.185,Y -449.022,Z 1946.515,A 0.000,B 0.000,C 90.000,E1 92.751} C_DIS
LIN {X 0.210,Y -448.935,Z 1946.512,A 0.000,B 0.000,C 90.000,E1 92.178} C_DIS
LIN {X 0.176,Y -447.901,Z 1946.509,A 0.000,B 0.000,C 90.000,E1 91.661} C_DIS
LIN {X 0.127,Y -445.749,Z 1946.506,A 0.000,B 0.000,C 90.000,E1 91.146} C_DIS
LIN {X 0.073,Y -434.307,Z 1946.496,A 0.000,B 0.000,C 90.000,E1 89.312} C_DIS
LIN {X 0.098,Y -424.300,Z 1946.487,A 0.000,B 0.000,C 90.000,E1 87.707} C_DIS
LIN {X 0.071,Y -412.513,Z 1946.477,A 0.000,B 0.000,C 90.000,E1 85.812} C_DIS
LIN {X 0.146,Y -402.357,Z 1946.468,A 0.000,B 0.000,C 90.000,E1 84.147} C_DIS
LIN {X 0.129,Y -390.370,Z 1946.457,A 0.000,B 0.000,C 90.000,E1 82.186} C_DIS
LIN {X -0.012,Y -378.489,Z 1946.446,A 0.000,B 0.000,C 90.000,E1 80.208} C_DIS
LIN {X -0.039,Y -365.131,Z 1946.433,A 0.000,B 0.000,C 90.000,E1 77.881} C_DIS
LIN {X 0.086,Y -347.799,Z 1946.414,A 0.000,B 0.000,C 90.000,E1 74.574} C_DIS
LIN {X 0.066,Y -334.354,Z 1946.399,A 0.000,B 0.000,C 90.000,E1 71.819} C_DIS
LIN {X -0.065,Y -322.669,Z 1946.385,A 0.000,B 0.000,C 90.000,E1 69.337} C_DIS
LIN {X 0.115,Y -308.693,Z 1946.367,A 0.000,B 0.000,C 90.000,E1 66.102} C_DIS
LIN {X 0.059,Y -300.585,Z 1946.356,A 0.000,B 0.000,C 90.000,E1 64.152} C_DIS
LIN {X -0.046,Y -288.540,Z 1946.340,A 0.000,B 0.000,C 90.000,E1 61.179} C_DIS
LIN {X 0.065,Y -280.483,Z 1946.328,A 0.000,B 0.000,C 90.000,E1 59.125} C_DIS
LIN {X 0.101,Y -270.937,Z 1946.315,A 0.000,B 0.000,C 90.000,E1 56.707} C_DIS
LIN {X 0.088,Y -262.686,Z 1946.303,A 0.000,B 0.000,C 90.000,E1 54.609} C_DIS
LIN {X -0.017,Y -251.704,Z 1946.288,A 0.000,B 0.000,C 90.000,E1 51.778} C_DIS
LIN {X 0.034,Y -242.136,Z 1946.273,A 0.000,B 0.000,C 90.000,E1 49.218} C_DIS
LIN {X -0.009,Y -231.545,Z 1946.257,A 0.000,B 0.000,C 90.000,E1 46.257} C_DIS
LIN {X 0.003,Y -221.297,Z 1946.240,A 0.000,B 0.000,C 90.000,E1 43.218} C_DIS
LIN {X 0.002,Y -210.476,Z 1946.221,A 0.000,B 0.000,C 90.000,E1 39.725} C_DIS
LIN {X -0.100,Y -201.696,Z 1946.203,A 0.000,B 0.000,C 90.000,E1 36.583} C_DIS
LIN {X 0.125,Y -193.742,Z 1946.185,A 0.000,B 0.000,C 90.000,E1 33.293} C_DIS
LIN {X -0.008,Y -186.511,Z 1946.167,A 0.000,B 0.000,C 90.000,E1 30.050} C_DIS
LIN {X -0.100,Y -180.045,Z 1946.148,A 0.000,B 0.000,C 90.000,E1 26.744} C_DIS
LIN {X -0.086,Y -175.656,Z 1946.134,A 0.000,B 0.000,C 90.000,E1 24.207} C_DIS
LIN {X 0.070,Y -170.542,Z 1946.115,A 0.000,B 0.000,C 90.000,E1 20.737} C_DIS
LIN {X 0.077,Y -166.263,Z 1946.096,A 0.000,B 0.000,C 90.000,E1 17.275} C_DIS
LIN {X -0.021,Y -161.983,Z 1946.072,A 0.000,B 0.000,C 90.000,E1 12.939} C_DIS
LIN {X 0.071,Y -159.257,Z 1946.052,A 0.000,B 0.000,C 90.000,E1 9.378} C_DIS
LIN {X -0.008,Y -156.505,Z 1946.023,A 0.000,B 0.000,C 90.000,E1 4.073} C_DIS
LIN {X -0.010,Y -154.435,Z 1945.982,A 0.000,B 0.000,C 90.000,E1 356.846} C_DIS
LIN {X 0.001,Y -155.583,Z 1945.918,A 0.000,B 0.000,C 90.000,E1 345.172} C_DIS
LIN {X -0.048,Y -158.033,Z 1945.888,A 0.000,B 0.000,C 90.000,E1 339.826} C_DIS
LIN {X 0.027,Y -161.377,Z 1945.863,A 0.000,B 0.000,C 90.000,E1 335.357} C_DIS
LIN {X -0.020,Y -164.979,Z 1945.844,A 0.000,B 0.000,C 90.000,E1 331.847} C_DIS
LIN {X 0.047,Y -169.594,Z 1945.824,A 0.000,B 0.000,C 90.000,E1 328.329} C_DIS
LIN {X -0.018,Y -173.670,Z 1945.810,A 0.000,B 0.000,C 90.000,E1 325.754} C_DIS
LIN {X 0.003,Y -178.377,Z 1945.795,A 0.000,B 0.000,C 90.000,E1 323.176} C_DIS
LIN {X -0.029,Y -183.928,Z 1945.781,A 0.000,B 0.000,C 90.000,E1 320.642} C_DIS
LIN {X 0.043,Y -189.237,Z 1945.770,A 0.000,B 0.000,C 90.000,E1 318.528} C_DIS
LIN {X 0.060,Y -195.320,Z 1945.758,A 0.000,B 0.000,C 90.000,E1 316.458} C_DIS
LIN {X 0.028,Y -203.450,Z 1945.745,A 0.000,B 0.000,C 90.000,E1 314.028} C_DIS
LIN {X 0.058,Y -214.052,Z 1945.729,A 0.000,B 0.000,C 90.000,E1 311.229} C_DIS
LIN {X -0.105,Y -225.721,Z 1945.714,A 0.000,B 0.000,C 90.000,E1 308.543} C_DIS
LIN {X 0.048,Y -240.231,Z 1945.697,A 0.000,B 0.000,C 90.000,E1 305.471} C_DIS
LIN {X -0.035,Y -255.810,Z 1945.681,A 0.000,B 0.000,C 90.000,E1 302.546} C_DIS
LIN {X 0.023,Y -267.819,Z 1945.669,A 0.000,B 0.000,C 90.000,E1 300.384} C_DIS
LIN {X 0.105,Y -277.842,Z 1945.659,A 0.000,B 0.000,C 90.000,E1 298.615} C_DIS
LIN {X -0.039,Y -287.583,Z 1945.650,A 0.000,B 0.000,C 90.000,E1 296.924} C_DIS
LIN {X 0.116,Y -295.012,Z 1945.642,A 0.000,B 0.000,C 90.000,E1 295.540} C_DIS
LIN {X -0.041,Y -300.039,Z 1945.636,A 0.000,B 0.000,C 90.000,E1 294.567} C_DIS
LIN {X -0.014,Y -303.020,Z 1945.633,A 0.000,B 0.000,C 90.000,E1 293.898} C_DIS
LIN {X 0.050,Y -306.777,Z 1945.627,A 0.000,B 0.000,C 90.000,E1 292.898} C_DIS
LIN {X -0.037,Y -308.785,Z 1945.624,A 0.000,B 0.000,C 90.000,E1 292.259} C_DIS
LIN {X 0.050,Y -310.444,Z 1945.620,A 0.000,B 0.000,C 90.000,E1 291.589} C_DIS
LIN {X 0.155,Y -311.784,Z 1945.616,A 0.000,B 0.000,C 90.000,E1 290.918} C_DIS
LIN {X -0.023,Y -312.775,Z 1945.613,A 0.000,B 0.000,C 90.000,E1 290.301} C_DIS
LIN {X 0.101,Y -313.428,Z 1945.609,A 0.000,B 0.000,C 90.000,E1 289.631} C_DIS
LIN {X -0.066,Y -313.771,Z 1945.606,A 0.000,B 0.000,C 90.000,E1 289.014} C_DIS
LIN {X -0.034,Y -313.760,Z 1945.602,A 0.000,B 0.000,C 90.000,E1 288.362} C_DIS
LIN {X 0.100,Y -313.371,Z 1945.598,A 0.000,B 0.000,C 90.000,E1 287.692} C_DIS
LIN {X 0.138,Y -312.540,Z 1945.595,A 0.000,B 0.000,C 90.000,E1 287.040} C_DIS
LIN {X -0.122,Y -311.225,Z 1945.591,A 0.000,B 0.000,C 90.000,E1 286.441} C_DIS
LIN {X -0.088,Y -309.407,Z 1945.588,A 0.000,B 0.000,C 90.000,E1 285.788} C_DIS
LIN {X -0.061,Y -306.935,Z 1945.584,A 0.000,B 0.000,C 90.000,E1 285.134} C_DIS
LIN {X -0.053,Y -303.701,Z 1945.580,A 0.000,B 0.000,C 90.000,E1 284.481} C_DIS
LIN {X 0.030,Y -297.746,Z 1945.575,A 0.000,B 0.000,C 90.000,E1 283.480} C_DIS
LIN {X -0.091,Y -292.655,Z 1945.570,A 0.000,B 0.000,C 90.000,E1 282.535} C_DIS
LIN {X 0.111,Y -288.700,Z 1945.566,A 0.000,B 0.000,C 90.000,E1 281.827} C_DIS
LIN {X -0.053,Y -283.880,Z 1945.562,A 0.000,B 0.000,C 90.000,E1 281.186} C_DIS
LIN {X -0.008,Y -281.057,Z 1945.560,A 0.000,B 0.000,C 90.000,E1 280.838} C_DIS
LIN {X -0.008,Y -274.872,Z 1945.557,A 0.000,B 0.000,C 90.000,E1 280.197} C_DIS
LIN {X 0.056,Y -268.437,Z 1945.553,A 0.000,B 0.000,C 90.000,E1 279.613} C_DIS
LIN {X 0.108,Y -261.794,Z 1945.551,A 0.000,B 0.000,C 90.000,E1 279.095} C_DIS
LIN {X -0.046,Y -255.079,Z 1945.548,A 0.000,B 0.000,C 90.000,E1 278.681} C_DIS
LIN {X 0.012,Y -248.134,Z 1945.546,A 0.000,B 0.000,C 90.000,E1 278.276} C_DIS
LIN {X 0.069,Y -240.701,Z 1945.544,A 0.000,B 0.000,C 90.000,E1 277.936} C_DIS
LIN {X -0.031,Y -232.620,Z 1945.543,A 0.000,B 0.000,C 90.000,E1 277.701} C_DIS
LIN {X -0.113,Y -222.155,Z 1945.542,A 0.000,B 0.000,C 90.000,E1 277.530} C_DIS
LIN {X -0.088,Y -212.222,Z 1945.541,A 0.000,B 0.000,C 90.000,E1 277.466} C_DIS
LIN {X 0.073,Y -180.205,Z 1945.541,A 0.000,B 0.000,C 90.000,E1 277.409} C_DIS
LIN {X 0.040,Y -181.029,Z 1945.530,A 0.000,B 0.000,C 90.000,E1 275.391} C_DIS
LIN {X 0.015,Y -181.579,Z 1945.502,A 0.000,B 0.000,C 90.000,E1 270.344} C_DIS
LIN {X -0.009,Y -180.904,Z 1945.474,A 0.000,B 0.000,C 90.000,E1 265.298} C_DIS
LIN {X -0.059,Y -180.242,Z 1945.464,A 0.000,B 0.000,C 90.000,E1 263.628} C_DIS
LIN {X -0.040,Y -178.729,Z 1945.441,A 0.000,B 0.000,C 90.000,E1 259.398} C_DIS
LIN {X 0.027,Y -175.777,Z 1945.413,A 0.000,B 0.000,C 90.000,E1 254.283} C_DIS
LIN {X 0.015,Y -171.961,Z 1945.384,A 0.000,B 0.000,C 90.000,E1 249.156} C_DIS
LIN {X 0.052,Y -171.355,Z 1945.379,A 0.000,B 0.000,C 90.000,E1 248.284} C_DIS
LIN {X 0.030,Y -167.605,Z 1945.355,A 0.000,B 0.000,C 90.000,E1 243.973} C_DIS
LIN {X 0.042,Y -166.250,Z 1945.346,A 0.000,B 0.000,C 90.000,E1 242.231} C_DIS
LIN {X 0.030,Y -163.006,Z 1945.326,A 0.000,B 0.000,C 90.000,E1 238.742} C_DIS
LIN {X 0.076,Y -160.929,Z 1945.312,A 0.000,B 0.000,C 90.000,E1 236.087} C_DIS
LIN {X 0.053,Y -157.689,Z 1945.292,A 0.000,B 0.000,C 90.000,E1 232.557} C_DIS
LIN {X -0.009,Y -155.729,Z 1945.277,A 0.000,B 0.000,C 90.000,E1 229.908} C_DIS
LIN {X 0.045,Y -151.988,Z 1945.252,A 0.000,B 0.000,C 90.000,E1 225.405} C_DIS
LIN {X 0.061,Y -150.232,Z 1945.237,A 0.000,B 0.000,C 90.000,E1 222.690} C_DIS
LIN {X -0.016,Y -146.993,Z 1945.212,A 0.000,B 0.000,C 90.000,E1 218.177} C_DIS
LIN {X -0.026,Y -145.578,Z 1945.197,A 0.000,B 0.000,C 90.000,E1 215.438} C_DIS
LIN {X -0.031,Y -142.968,Z 1945.171,A 0.000,B 0.000,C 90.000,E1 210.846} C_DIS
LIN {X 0.022,Y -141.594,Z 1945.151,A 0.000,B 0.000,C 90.000,E1 207.129} C_DIS
LIN {X 0.068,Y -139.421,Z 1945.115,A 0.000,B 0.000,C 90.000,E1 200.610} C_DIS
LIN {X -0.011,Y -139.148,Z 1945.104,A 0.000,B 0.000,C 90.000,E1 198.779} C_DIS
LIN {X 0.011,Y -138.346,Z 1945.058,A 0.000,B 0.000,C 90.000,E1 190.366} C_DIS
LIN {X -0.003,Y -139.488,Z 1945.006,A 0.000,B 0.000,C 90.000,E1 181.031} C_DIS
LIN {X -0.063,Y -141.090,Z 1944.975,A 0.000,B 0.000,C 90.000,E1 175.469} C_DIS
LIN {X 0.031,Y -142.467,Z 1944.959,A 0.000,B 0.000,C 90.000,E1 172.648} C_DIS
LIN {X -0.021,Y -144.713,Z 1944.934,A 0.000,B 0.000,C 90.000,E1 168.049} C_DIS
LIN {X -0.069,Y -147.313,Z 1944.913,A 0.000,B 0.000,C 90.000,E1 164.393} C_DIS
LIN {X -0.055,Y -150.633,Z 1944.888,A 0.000,B 0.000,C 90.000,E1 159.826} C_DIS
LIN {X 0.021,Y -154.110,Z 1944.868,A 0.000,B 0.000,C 90.000,E1 156.177} C_DIS
LIN {X -0.056,Y -157.534,Z 1944.848,A 0.000,B 0.000,C 90.000,E1 152.615} C_DIS
LIN {X -0.028,Y -161.771,Z 1944.828,A 0.000,B 0.000,C 90.000,E1 149.046} C_DIS
LIN {X -0.006,Y -165.963,Z 1944.808,A 0.000,B 0.000,C 90.000,E1 145.515} C_DIS
LIN {X -0.010,Y -170.957,Z 1944.789,A 0.000,B 0.000,C 90.000,E1 142.029} C_DIS
LIN {X 0.042,Y -175.826,Z 1944.770,A 0.000,B 0.000,C 90.000,E1 138.566} C_DIS
LIN {X 0.037,Y -181.433,Z 1944.751,A 0.000,B 0.000,C 90.000,E1 135.162} C_DIS
LIN {X -0.089,Y -186.938,Z 1944.732,A 0.000,B 0.000,C 90.000,E1 131.838} C_DIS
LIN {X -0.090,Y -190.049,Z 1944.723,A 0.000,B 0.000,C 90.000,E1 130.172} C_DIS
LIN {X -0.075,Y -195.825,Z 1944.705,A 0.000,B 0.000,C 90.000,E1 126.870} C_DIS
LIN {X -0.008,Y -200.657,Z 1944.691,A 0.000,B 0.000,C 90.000,E1 124.405} C_DIS
LIN {X 0.009,Y -206.541,Z 1944.673,A 0.000,B 0.000,C 90.000,E1 121.180} C_DIS
LIN {X -0.004,Y -209.832,Z 1944.664,A 0.000,B 0.000,C 90.000,E1 119.589} C_DIS
LIN {X -0.079,Y -217.190,Z 1944.642,A 0.000,B 0.000,C 90.000,E1 115.668} C_DIS
LIN {X -0.124,Y -218.817,Z 1944.638,A 0.000,B 0.000,C 90.000,E1 114.899} C_DIS
LIN {X 0.099,Y -224.203,Z 1944.621,A 0.000,B 0.000,C 90.000,E1 111.770} C_DIS
LIN {X 0.093,Y -283.984,Z 1944.621,A 0.000,B 0.000,C 90.000,E1 111.770} C_DIS
LIN {X -0.003,Y -285.277,Z 1944.621,A 0.000,B 0.000,C 90.000,E1 111.770} C_DIS
LIN {X -0.004,Y -288.621,Z 1944.620,A 0.000,B 0.000,C 90.000,E1 111.642} C_DIS
LIN {X -0.036,Y -291.870,Z 1944.619,A 0.000,B 0.000,C 90.000,E1 111.408} C_DIS
LIN {X -0.073,Y -295.549,Z 1944.616,A 0.000,B 0.000,C 90.000,E1 110.972} C_DIS
LIN {X -0.027,Y -312.780,Z 1944.600,A 0.000,B 0.000,C 90.000,E1 108.000} C_DIS
LIN {X 0.058,Y -327.708,Z 1944.587,A 0.000,B 0.000,C 90.000,E1 105.733} C_DIS
LIN {X -0.142,Y -341.708,Z 1944.577,A 0.000,B 0.000,C 90.000,E1 103.883} C_DIS
LIN {X 0.097,Y -356.907,Z 1944.567,A 0.000,B 0.000,C 90.000,E1 102.007} C_DIS
LIN {X 0.068,Y -375.403,Z 1944.556,A 0.000,B 0.000,C 90.000,E1 100.018} C_DIS
LIN {X -0.046,Y -394.360,Z 1944.546,A 0.000,B 0.000,C 90.000,E1 98.219} C_DIS
LIN {X 0.151,Y -416.451,Z 1944.535,A 0.000,B 0.000,C 90.000,E1 96.315} C_DIS
LIN {X -0.015,Y -438.948,Z 1944.526,A 0.000,B 0.000,C 90.000,E1 94.645} C_DIS
LIN {X 0.005,Y -443.211,Z 1944.524,A 0.000,B 0.000,C 90.000,E1 94.245} C_DIS
LIN {X -0.175,Y -446.286,Z 1944.521,A 0.000,B 0.000,C 90.000,E1 93.784} C_DIS
LIN {X 0.185,Y -448.193,Z 1944.518,A 0.000,B 0.000,C 90.000,E1 93.212} C_DIS
LIN {X 0.143,Y -449.018,Z 1944.515,A 0.000,B 0.000,C 90.000,E1 92.694} C_DIS
LIN {X 0.089,Y -448.903,Z 1944.512,A 0.000,B 0.000,C 90.000,E1 92.178} C_DIS
LIN {X 0.056,Y -447.838,Z 1944.509,A 0.000,B 0.000,C 90.000,E1 91.661} C_DIS
LIN {X -0.192,Y -446.903,Z 1944.508,A 0.000,B 0.000,C 90.000,E1 91.432} C_DIS
LIN {X 0.007,Y -445.645,Z 1944.506,A 0.000,B 0.000,C 90.000,E1 91.146} C_DIS
LIN {X -0.051,Y -434.188,Z 1944.496,A 0.000,B 0.000,C 90.000,E1 89.312} C_DIS
LIN {X -0.025,Y -424.176,Z 1944.487,A 0.000,B 0.000,C 90.000,E1 87.707} C_DIS
LIN {X -0.052,Y -412.391,Z 1944.477,A 0.000,B 0.000,C 90.000,E1 85.812} C_DIS
LIN {X 0.025,Y -402.232,Z 1944.468,A 0.000,B 0.000,C 90.000,E1 84.147} C_DIS
LIN {X 0.009,Y -390.246,Z 1944.457,A 0.000,B 0.000,C 90.000,E1 82.186} C_DIS
LIN {X -0.131,Y -378.367,Z 1944.445,A 0.000,B 0.000,C 90.000,E1 80.208} C_DIS
LIN {X -0.157,Y -365.009,Z 1944.432,A 0.000,B 0.000,C 90.000,E1 77.881} C_DIS
LIN {X -0.030,Y -347.683,Z 1944.414,A 0.000,B 0.000,C 90.000,E1 74.574} C_DIS
LIN {X -0.049,Y -334.241,Z 1944.399,A 0.000,B 0.000,C 90.000,E1 71.819} C_DIS
LIN {X -0.064,Y -322.556,Z 1944.385,A 0.000,B 0.000,C 90.000,E1 69.316} C_DIS
LIN {X 0.003,Y -308.586,Z 1944.367,A 0.000,B 0.000,C 90.000,E1 66.102} C_DIS
LIN {X -0.053,Y -300.474,Z 1944.356,A 0.000,B 0.000,C 90.000,E1 64.152} C_DIS
LIN {X 0.098,Y -288.432,Z 1944.340,A 0.000,B 0.000,C 90.000,E1 61.129} C_DIS
LIN {X -0.044,Y -280.373,Z 1944.328,A 0.000,B 0.000,C 90.000,E1 59.125} C_DIS
LIN {X -0.007,Y -270.828,Z 1944.315,A 0.000,B 0.000,C 90.000,E1 56.707} C_DIS
LIN {X -0.018,Y -262.576,Z 1944.303,A 0.000,B 0.000,C 90.000,E1 54.609} C_DIS
LIN {X 0.002,Y -252.966,Z 1944.290,A 0.000,B 0.000,C 90.000,E1 52.110} C_DIS
LIN {X 0.119,Y -243.388,Z 1944.275,A 0.000,B 0.000,C 90.000,E1 49.542} C_DIS
LIN {X -0.060,Y -232.739,Z 1944.259,A 0.000,B 0.000,C 90.000,E1 46.620} C_DIS
LIN {X -0.017,Y -222.464,Z 1944.242,A 0.000,B 0.000,C 90.000,E1 43.581} C_DIS
LIN {X -0.002,Y -211.543,Z 1944.223,A 0.000,B 0.000,C 90.000,E1 40.092} C_DIS
LIN {X 0.029,Y -203.713,Z 1944.207,A 0.000,B 0.000,C 90.000,E1 37.317} C_DIS
LIN {X -0.017,Y -195.577,Z 1944.190,A 0.000,B 0.000,C 90.000,E1 34.119} C_DIS
LIN {X -0.001,Y -188.181,Z 1944.171,A 0.000,B 0.000,C 90.000,E1 30.846} C_DIS
LIN {X 0.032,Y -181.534,Z 1944.153,A 0.000,B 0.000,C 90.000,E1 27.513} C_DIS
LIN {X -0.092,Y -177.003,Z 1944.139,A 0.000,B 0.000,C 90.000,E1 25.027} C_DIS
LIN {X 0.005,Y -171.706,Z 1944.120,A 0.000,B 0.000,C 90.000,E1 21.589} C_DIS
LIN {X 0.040,Y -167.198,Z 1944.101,A 0.000,B 0.000,C 90.000,E1 18.127} C_DIS
LIN {X -0.019,Y -163.555,Z 1944.081,A 0.000,B 0.000,C 90.000,E1 14.662} C_DIS
LIN {X 0.009,Y -159.831,Z 1944.057,A 0.000,B 0.000,C 90.000,E1 10.254} C_DIS
LIN {X 0.071,Y -157.261,Z 1944.032,A 0.000,B 0.000,C 90.000,E1 5.796} C_DIS
LIN {X -0.028,Y -154.946,Z 1943.997,A 0.000,B 0.000,C 90.000,E1 359.542} C_DIS
LIN {X 0.059,Y -154.184,Z 1943.953,A 0.000,B 0.000,C 90.000,E1 351.432} C_DIS
LIN {X -0.018,Y -155.895,Z 1943.913,A 0.000,B 0.000,C 90.000,E1 344.283} C_DIS
LIN {X 0.046,Y -158.600,Z 1943.883,A 0.000,B 0.000,C 90.000,E1 338.901} C_DIS
LIN {X 0.062,Y -162.184,Z 1943.858,A 0.000,B 0.000,C 90.000,E1 334.460} C_DIS
LIN {X -0.032,Y -166.039,Z 1943.839,A 0.000,B 0.000,C 90.000,E1 330.973} C_DIS
LIN {X 0.065,Y -170.894,Z 1943.819,A 0.000,B 0.000,C 90.000,E1 327.454} C_DIS
LIN {X -0.023,Y -175.176,Z 1943.805,A 0.000,B 0.000,C 90.000,E1 324.895} C_DIS
LIN {X 0.029,Y -180.131,Z 1943.791,A 0.000,B 0.000,C 90.000,E1 322.316} C_DIS
LIN {X 0.026,Y -185.986,Z 1943.777,A 0.000,B 0.000,C 90.000,E1 319.784} C_DIS
LIN {X -0.009,Y -191.595,Z 1943.765,A 0.000,B 0.000,C 90.000,E1 317.715} C_DIS
LIN {X 0.026,Y -199.281,Z 1943.751,A 0.000,B 0.000,C 90.000,E1 315.243} C_DIS
LIN {X -0.072,Y -207.869,Z 1943.738,A 0.000,B 0.000,C 90.000,E1 312.852} C_DIS
LIN {X -0.094,Y -218.919,Z 1943.723,A 0.000,B 0.000,C 90.000,E1 310.092} C_DIS
LIN {X -0.030,Y -232.837,Z 1943.705,A 0.000,B 0.000,C 90.000,E1 306.996} C_DIS
LIN {X 0.030,Y -247.889,Z 1943.689,A 0.000,B 0.000,C 90.000,E1 303.992} C_DIS
LIN {X 0.079,Y -259.814,Z 1943.677,A 0.000,B 0.000,C 90.000,E1 301.799} C_DIS
LIN {X 0.082,Y -271.873,Z 1943.665,A 0.000,B 0.000,C 90.000,E1 299.667} C_DIS
LIN {X -0.146,Y -281.780,Z 1943.655,A 0.000,B 0.000,C 90.000,E1 297.975} C_DIS
LIN {X 0.025,Y -291.377,Z 1943.646,A 0.000,B 0.000,C 90.000,E1 296.232} C_DIS
LIN {X 0.105,Y -296.779,Z 1943.640,A 0.000,B 0.000,C 90.000,E1 295.207} C_DIS
LIN {X 0.105,Y -301.575,Z 1943.635,A 0.000,B 0.000,C 90.000,E1 294.207} C_DIS
LIN {X -0.010,Y -304.384,Z 1943.631,A 0.000,B 0.000,C 90.000,E1 293.567} C_DIS
LIN {X 0.051,Y -306.789,Z 1943.627,A 0.000,B 0.000,C 90.000,E1 292.898} C_DIS
LIN {X -0.036,Y -308.798,Z 1943.624,A 0.000,B 0.000,C 90.000,E1 292.259} C_DIS
LIN {X 0.052,Y -310.459,Z 1943.620,A 0.000,B 0.000,C 90.000,E1 291.589} C_DIS
LIN {X -0.136,Y -311.798,Z 1943.616,A 0.000,B 0.000,C 90.000,E1 290.972} C_DIS
LIN {X -0.021,Y -312.791,Z 1943.613,A 0.000,B 0.000,C 90.000,E1 290.301} C_DIS
LIN {X 0.102,Y -313.441,Z 1943.609,A 0.000,B 0.000,C 90.000,E1 289.631} C_DIS
LIN {X -0.065,Y -313.785,Z 1943.606,A 0.000,B 0.000,C 90.000,E1 289.014} C_DIS
LIN {X -0.032,Y -313.774,Z 1943.602,A 0.000,B 0.000,C 90.000,E1 288.362} C_DIS
LIN {X 0.102,Y -313.386,Z 1943.598,A 0.000,B 0.000,C 90.000,E1 287.692} C_DIS
LIN {X 0.140,Y -312.557,Z 1943.595,A 0.000,B 0.000,C 90.000,E1 287.040} C_DIS
LIN {X -0.120,Y -311.244,Z 1943.591,A 0.000,B 0.000,C 90.000,E1 286.441} C_DIS
LIN {X -0.086,Y -309.422,Z 1943.588,A 0.000,B 0.000,C 90.000,E1 285.788} C_DIS
LIN {X -0.059,Y -306.953,Z 1943.584,A 0.000,B 0.000,C 90.000,E1 285.134} C_DIS
LIN {X -0.051,Y -303.719,Z 1943.580,A 0.000,B 0.000,C 90.000,E1 284.481} C_DIS
LIN {X 0.032,Y -297.766,Z 1943.575,A 0.000,B 0.000,C 90.000,E1 283.480} C_DIS
LIN {X 0.067,Y -292.533,Z 1943.569,A 0.000,B 0.000,C 90.000,E1 282.479} C_DIS
LIN {X -0.016,Y -288.551,Z 1943.566,A 0.000,B 0.000,C 90.000,E1 281.827} C_DIS
LIN {X 0.101,Y -283.674,Z 1943.562,A 0.000,B 0.000,C 90.000,E1 281.130} C_DIS
LIN {X -0.131,Y -280.850,Z 1943.560,A 0.000,B 0.000,C 90.000,E1 280.838} C_DIS
LIN {X -0.118,Y -274.625,Z 1943.557,A 0.000,B 0.000,C 90.000,E1 280.197} C_DIS
LIN {X -0.038,Y -268.200,Z 1943.553,A 0.000,B 0.000,C 90.000,E1 279.613} C_DIS
LIN {X 0.028,Y -261.549,Z 1943.551,A 0.000,B 0.000,C 90.000,E1 279.095} C_DIS
LIN {X -0.107,Y -254.833,Z 1943.548,A 0.000,B 0.000,C 90.000,E1 278.681} C_DIS
LIN {X -0.041,Y -247.884,Z 1943.546,A 0.000,B 0.000,C 90.000,E1 278.276} C_DIS
LIN {X 0.025,Y -240.411,Z 1943.544,A 0.000,B 0.000,C 90.000,E1 277.936} C_DIS
LIN {X -0.063,Y -232.278,Z 1943.543,A 0.000,B 0.000,C 90.000,E1 277.701} C_DIS
LIN {X 0.084,Y -221.500,Z 1943.542,A 0.000,B 0.000,C 90.000,E1 277.473} C_DIS
LIN {X -0.071,Y -215.437,Z 1943.541,A 0.000,B 0.000,C 90.000,E1 277.466} C_DIS
LIN {X 0.089,Y -180.203,Z 1943.541,A 0.000,B 0.000,C 90.000,E1 277.409} C_DIS
LIN {X 0.026,Y -181.029,Z 1943.530,A 0.000,B 0.000,C 90.000,E1 275.391} C_DIS
LIN {X 0.001,Y -181.579,Z 1943.502,A 0.000,B 0.000,C 90.000,E1 270.344} C_DIS
LIN {X -0.023,Y -180.904,Z 1943.474,A 0.000,B 0.000,C 90.000,E1 265.298} C_DIS
LIN {X -0.073,Y -180.241,Z 1943.464,A 0.000,B 0.000,C 90.000,E1 263.628} C_DIS
LIN {X -0.055,Y -178.726,Z 1943.441,A 0.000,B 0.000,C 90.000,E1 259.398} C_DIS
LIN {X 0.013,Y -175.775,Z 1943.413,A 0.000,B 0.000,C 90.000,E1 254.283} C_DIS
LIN {X 0.001,Y -171.958,Z 1943.384,A 0.000,B 0.000,C 90.000,E1 249.156} C_DIS
LIN {X 0.038,Y -171.351,Z 1943.379,A 0.000,B 0.000,C 90.000,E1 248.284} C_DIS
LIN {X 0.016,Y -167.602,Z 1943.355,A 0.000,B 0.000,C 90.000,E1 243.973} C_DIS
LIN {X 0.029,Y -166.246,Z 1943.346,A 0.000,B 0.000,C 90.000,E1 242.231} C_DIS
LIN {X 0.016,Y -163.003,Z 1943.326,A 0.000,B 0.000,C 90.000,E1 238.742} C_DIS
LIN {X 0.063,Y -160.923,Z 1943.312,A 0.000,B 0.000,C 90.000,E1 236.087} C_DIS
LIN {X 0.041,Y -157.686,Z 1943.292,A 0.000,B 0.000,C 90.000,E1 232.557} C_DIS
LIN {X -0.021,Y -155.725,Z 1943.277,A 0.000,B 0.000,C 90.000,E1 229.908} C_DIS
LIN {X 0.033,Y -151.984,Z 1943.252,A 0.000,B 0.000,C 90.000,E1 225.405} C_DIS
LIN {X 0.048,Y -150.228,Z 1943.237,A 0.000,B 0.000,C 90.000,E1 222.690} C_DIS
LIN {X -0.029,Y -146.990,Z 1943.212,A 0.000,B 0.000,C 90.000,E1 218.177} C_DIS
LIN {X -0.038,Y -145.576,Z 1943.197,A 0.000,B 0.000,C 90.000,E1 215.438} C_DIS
LIN {X 0.079,Y -142.965,Z 1943.171,A 0.000,B 0.000,C 90.000,E1 210.797} C_DIS
LIN {X 0.009,Y -141.592,Z 1943.151,A 0.000,B 0.000,C 90.000,E1 207.129} C_DIS
LIN {X 0.057,Y -139.420,Z 1943.115,A 0.000,B 0.000,C 90.000,E1 200.610} C_DIS
LIN {X -0.023,Y -139.147,Z 1943.104,A 0.000,B 0.000,C 90.000,E1 198.779} C_DIS
LIN {X -0.001,Y -138.346,Z 1943.058,A 0.000,B 0.000,C 90.000,E1 190.366} C_DIS
LIN {X -0.015,Y -139.488,Z 1943.006,A 0.000,B 0.000,C 90.000,E1 181.031} C_DIS
LIN {X 0.065,Y -141.092,Z 1942.975,A 0.000,B 0.000,C 90.000,E1 175.412} C_DIS
LIN {X 0.019,Y -142.470,Z 1942.959,A 0.000,B 0.000,C 90.000,E1 172.648} C_DIS
LIN {X -0.033,Y -144.716,Z 1942.934,A 0.000,B 0.000,C 90.000,E1 168.049} C_DIS
LIN {X 0.060,Y -147.316,Z 1942.913,A 0.000,B 0.000,C 90.000,E1 164.338} C_DIS
LIN {X -0.015,Y -150.638,Z 1942.888,A 0.000,B 0.000,C 90.000,E1 159.806} C_DIS
LIN {X 0.008,Y -154.114,Z 1942.868,A 0.000,B 0.000,C 90.000,E1 156.177} C_DIS
LIN {X -0.068,Y -157.540,Z 1942.848,A 0.000,B 0.000,C 90.000,E1 152.615} C_DIS
LIN {X 0.097,Y -161.778,Z 1942.828,A 0.000,B 0.000,C 90.000,E1 148.997} C_DIS
LIN {X -0.019,Y -165.970,Z 1942.808,A 0.000,B 0.000,C 90.000,E1 145.515} C_DIS
LIN {X -0.024,Y -170.964,Z 1942.789,A 0.000,B 0.000,C 90.000,E1 142.029} C_DIS
LIN {X 0.028,Y -175.833,Z 1942.770,A 0.000,B 0.000,C 90.000,E1 138.566} C_DIS
LIN {X 0.023,Y -181.439,Z 1942.751,A 0.000,B 0.000,C 90.000,E1 135.162} C_DIS
LIN {X -0.104,Y -186.946,Z 1942.732,A 0.000,B 0.000,C 90.000,E1 131.838} C_DIS
LIN {X -0.104,Y -190.058,Z 1942.723,A 0.000,B 0.000,C 90.000,E1 130.172} C_DIS
LIN {X -0.090,Y -195.833,Z 1942.705,A 0.000,B 0.000,C 90.000,E1 126.870} C_DIS
LIN {X -0.023,Y -200.665,Z 1942.691,A 0.000,B 0.000,C 90.000,E1 124.405} C_DIS
LIN {X -0.007,Y -206.549,Z 1942.673,A 0.000,B 0.000,C 90.000,E1 121.180} C_DIS
LIN {X -0.020,Y -209.841,Z 1942.664,A 0.000,B 0.000,C 90.000,E1 119.589} C_DIS
LIN {X 0.000,Y -217.199,Z 1942.642,A 0.000,B 0.000,C 90.000,E1 115.643} C_DIS
LIN {X 0.058,Y -218.826,Z 1942.638,A 0.000,B 0.000,C 90.000,E1 114.847} C_DIS
LIN {X 0.110,Y -224.198,Z 1942.621,A 0.000,B 0.000,C 90.000,E1 111.770} C_DIS
LIN {X 0.107,Y -283.827,Z 1942.621,A 0.000,B 0.000,C 90.000,E1 111.770} C_DIS
LIN {X -0.023,Y -285.519,Z 1942.621,A 0.000,B 0.000,C 90.000,E1 111.770} C_DIS
LIN {X -0.078,Y -288.524,Z 1942.620,A 0.000,B 0.000,C 90.000,E1 111.663} C_DIS
LIN {X -0.028,Y -291.861,Z 1942.619,A 0.000,B 0.000,C 90.000,E1 111.408} C_DIS
LIN {X -0.052,Y -295.524,Z 1942.616,A 0.000,B 0.000,C 90.000,E1 110.972} C_DIS
LIN {X -0.004,Y -312.752,Z 1942.600,A 0.000,B 0.000,C 90.000,E1 108.000} C_DIS
LIN {X 0.082,Y -327.676,Z 1942.588,A 0.000,B 0.000,C 90.000,E1 105.733} C_DIS
LIN {X -0.117,Y -341.674,Z 1942.577,A 0.000,B 0.000,C 90.000,E1 103.883} C_DIS
LIN {X 0.122,Y -356.872,Z 1942.567,A 0.000,B 0.000,C 90.000,E1 102.007} C_DIS
LIN {X 0.091,Y -375.366,Z 1942.556,A 0.000,B 0.000,C 90.000,E1 100.018} C_DIS
LIN {X -0.025,Y -394.323,Z 1942.546,A 0.000,B 0.000,C 90.000,E1 98.219} C_DIS
LIN {X 0.173,Y -416.412,Z 1942.535,A 0.000,B 0.000,C 90.000,E1 96.315} C_DIS
LIN {X 0.005,Y -438.910,Z 1942.526,A 0.000,B 0.000,C 90.000,E1 94.645} C_DIS
LIN {X 0.025,Y -443.184,Z 1942.524,A 0.000,B 0.000,C 90.000,E1 94.245} C_DIS
LIN {X -0.150,Y -446.260,Z 1942.521,A 0.000,B 0.000,C 90.000,E1 93.784} C_DIS
LIN {X 0.210,Y -448.172,Z 1942.518,A 0.000,B 0.000,C 90.000,E1 93.212} C_DIS
LIN {X 0.167,Y -449.001,Z 1942.515,A 0.000,B 0.000,C 90.000,E1 92.694} C_DIS
LIN {X 0.113,Y -448.891,Z 1942.512,A 0.000,B 0.000,C 90.000,E1 92.178} C_DIS
LIN {X 0.080,Y -447.830,Z 1942.509,A 0.000,B 0.000,C 90.000,E1 91.661} C_DIS
LIN {X -0.167,Y -446.897,Z 1942.508,A 0.000,B 0.000,C 90.000,E1 91.432} C_DIS
LIN {X 0.032,Y -445.644,Z 1942.506,A 0.000,B 0.000,C 90.000,E1 91.146} C_DIS
LIN {X -0.027,Y -434.189,Z 1942.496,A 0.000,B 0.000,C 90.000,E1 89.312} C_DIS
LIN {X -0.001,Y -424.176,Z 1942.487,A 0.000,B 0.000,C 90.000,E1 87.707} C_DIS
LIN {X -0.030,Y -412.391,Z 1942.477,A 0.000,B 0.000,C 90.000,E1 85.812} C_DIS
LIN {X 0.047,Y -402.234,Z 1942.468,A 0.000,B 0.000,C 90.000,E1 84.147} C_DIS
LIN {X 0.031,Y -390.248,Z 1942.457,A 0.000,B 0.000,C 90.000,E1 82.186} C_DIS
LIN {X -0.110,Y -378.366,Z 1942.446,A 0.000,B 0.000,C 90.000,E1 80.208} C_DIS
LIN {X -0.136,Y -365.008,Z 1942.432,A 0.000,B 0.000,C 90.000,E1 77.881} C_DIS
LIN {X -0.011,Y -347.680,Z 1942.414,A 0.000,B 0.000,C 90.000,E1 74.574} C_DIS
LIN {X -0.031,Y -334.236,Z 1942.399,A 0.000,B 0.000,C 90.000,E1 71.819} C_DIS
LIN {X -0.048,Y -322.550,Z 1942.385,A 0.000,B 0.000,C 90.000,E1 69.316} C_DIS
LIN {X 0.019,Y -308.578,Z 1942.367,A 0.000,B 0.000,C 90.000,E1 66.102} C_DIS
LIN {X -0.036,Y -300.464,Z 1942.356,A 0.000,B 0.000,C 90.000,E1 64.152} C_DIS
LIN {X -0.139,Y -288.421,Z 1942.340,A 0.000,B 0.000,C 90.000,E1 61.179} C_DIS
LIN {X -0.029,Y -280.362,Z 1942.328,A 0.000,B 0.000,C 90.000,E1 59.125} C_DIS
LIN {X 0.007,Y -270.820,Z 1942.315,A 0.000,B 0.000,C 90.000,E1 56.707} C_DIS
LIN {X -0.006,Y -262.570,Z 1942.303,A 0.000,B 0.000,C 90.000,E1 54.609} C_DIS
LIN {X 0.015,Y -252.961,Z 1942.290,A 0.000,B 0.000,C 90.000,E1 52.110} C_DIS
LIN {X -0.054,Y -243.383,Z 1942.275,A 0.000,B 0.000,C 90.000,E1 49.585} C_DIS
LIN {X -0.049,Y -232.732,Z 1942.259,A 0.000,B 0.000,C 90.000,E1 46.620} C_DIS
LIN {X -0.007,Y -222.456,Z 1942.242,A 0.000,B 0.000,C 90.000,E1 43.581} C_DIS
LIN {X 0.008,Y -211.535,Z 1942.223,A 0.000,B 0.000,C 90.000,E1 40.092} C_DIS
LIN {X 0.038,Y -203.705,Z 1942.207,A 0.000,B 0.000,C 90.000,E1 37.317} C_DIS
LIN {X -0.008,Y -195.571,Z 1942.190,A 0.000,B 0.000,C 90.000,E1 34.119} C_DIS
LIN {X 0.008,Y -188.178,Z 1942.171,A 0.000,B 0.000,C 90.000,E1 30.846} C_DIS
LIN {X 0.039,Y -181.530,Z 1942.153,A 0.000,B 0.000,C 90.000,E1 27.513} C_DIS
LIN {X -0.006,Y -175.598,Z 1942.134,A 0.000,B 0.000,C 90.000,E1 24.155} C_DIS
LIN {X -0.010,Y -170.492,Z 1942.115,A 0.000,B 0.000,C 90.000,E1 20.737} C_DIS
LIN {X -0.002,Y -166.221,Z 1942.096,A 0.000,B 0.000,C 90.000,E1 17.275} C_DIS
LIN {X 0.058,Y -161.944,Z 1942.072,A 0.000,B 0.000,C 90.000,E1 12.883} C_DIS
LIN {X -0.007,Y -159.224,Z 1942.052,A 0.000,B 0.000,C 90.000,E1 9.378} C_DIS
LIN {X 0.082,Y -156.477,Z 1942.022,A 0.000,B 0.000,C 90.000,E1 4.012} C_DIS
LIN {X -0.011,Y -154.415,Z 1941.982,A 0.000,B 0.000,C 90.000,E1 356.846} C_DIS
LIN {X -0.001,Y -155.572,Z 1941.918,A 0.000,B 0.000,C 90.000,E1 345.172} C_DIS
LIN {X -0.050,Y -158.025,Z 1941.888,A 0.000,B 0.000,C 90.000,E1 339.826} C_DIS
LIN {X 0.025,Y -161.374,Z 1941.863,A 0.000,B 0.000,C 90.000,E1 335.357} C_DIS
LIN {X -0.022,Y -164.982,Z 1941.844,A 0.000,B 0.000,C 90.000,E1 331.847} C_DIS
LIN {X 0.045,Y -169.604,Z 1941.824,A 0.000,B 0.000,C 90.000,E1 328.329} C_DIS
LIN {X -0.020,Y -173.683,Z 1941.810,A 0.000,B 0.000,C 90.000,E1 325.754} C_DIS
LIN {X 0.000,Y -178.393,Z 1941.795,A 0.000,B 0.000,C 90.000,E1 323.176} C_DIS
LIN {X -0.031,Y -183.947,Z 1941.781,A 0.000,B 0.000,C 90.000,E1 320.642} C_DIS
LIN {X 0.041,Y -189.256,Z 1941.770,A 0.000,B 0.000,C 90.000,E1 318.528} C_DIS
LIN {X 0.059,Y -195.335,Z 1941.758,A 0.000,B 0.000,C 90.000,E1 316.458} C_DIS
LIN {X 0.027,Y -203.461,Z 1941.745,A 0.000,B 0.000,C 90.000,E1 314.028} C_DIS
LIN {X 0.058,Y -214.067,Z 1941.729,A 0.000,B 0.000,C 90.000,E1 311.229} C_DIS
LIN {X -0.105,Y -225.735,Z 1941.714,A 0.000,B 0.000,C 90.000,E1 308.543} C_DIS
LIN {X 0.048,Y -240.252,Z 1941.697,A 0.000,B 0.000,C 90.000,E1 305.471} C_DIS
LIN {X -0.034,Y -255.831,Z 1941.681,A 0.000,B 0.000,C 90.000,E1 302.546} C_DIS
LIN {X 0.024,Y -267.837,Z 1941.669,A 0.000,B 0.000,C 90.000,E1 300.384} C_DIS
LIN {X 0.107,Y -277.862,Z 1941.659,A 0.000,B 0.000,C 90.000,E1 298.615} C_DIS
LIN {X -0.037,Y -287.602,Z 1941.650,A 0.000,B 0.000,C 90.000,E1 296.924} C_DIS
LIN {X 0.117,Y -295.030,Z 1941.642,A 0.000,B 0.000,C 90.000,E1 295.540} C_DIS
LIN {X -0.038,Y -300.062,Z 1941.636,A 0.000,B 0.000,C 90.000,E1 294.567} C_DIS
LIN {X -0.009,Y -304.396,Z 1941.631,A 0.000,B 0.000,C 90.000,E1 293.567} C_DIS
LIN {X 0.052,Y -306.802,Z 1941.627,A 0.000,B 0.000,C 90.000,E1 292.898} C_DIS
LIN {X -0.034,Y -308.811,Z 1941.624,A 0.000,B 0.000,C 90.000,E1 292.259} C_DIS
LIN {X 0.053,Y -310.473,Z 1941.620,A 0.000,B 0.000,C 90.000,E1 291.589} C_DIS
LIN {X -0.134,Y -311.813,Z 1941.616,A 0.000,B 0.000,C 90.000,E1 290.972} C_DIS
LIN {X -0.020,Y -312.807,Z 1941.613,A 0.000,B 0.000,C 90.000,E1 290.301} C_DIS
LIN {X 0.104,Y -313.454,Z 1941.609,A 0.000,B 0.000,C 90.000,E1 289.631} C_DIS
LIN {X -0.063,Y -313.799,Z 1941.606,A 0.000,B 0.000,C 90.000,E1 289.014} C_DIS
LIN {X -0.031,Y -313.789,Z 1941.602,A 0.000,B 0.000,C 90.000,E1 288.362} C_DIS
LIN {X 0.104,Y -313.401,Z 1941.598,A 0.000,B 0.000,C 90.000,E1 287.692} C_DIS
LIN {X 0.142,Y -312.576,Z 1941.595,A 0.000,B 0.000,C 90.000,E1 287.040} C_DIS
LIN {X -0.118,Y -311.263,Z 1941.591,A 0.000,B 0.000,C 90.000,E1 286.441} C_DIS
LIN {X -0.083,Y -309.438,Z 1941.588,A 0.000,B 0.000,C 90.000,E1 285.788} C_DIS
LIN {X -0.057,Y -306.972,Z 1941.584,A 0.000,B 0.000,C 90.000,E1 285.134} C_DIS
LIN {X -0.048,Y -303.738,Z 1941.580,A 0.000,B 0.000,C 90.000,E1 284.481} C_DIS
LIN {X -0.092,Y -295.995,Z 1941.573,A 0.000,B 0.000,C 90.000,E1 283.175} C_DIS
LIN {X 0.070,Y -292.548,Z 1941.569,A 0.000,B 0.000,C 90.000,E1 282.479} C_DIS
LIN {X -0.013,Y -288.563,Z 1941.566,A 0.000,B 0.000,C 90.000,E1 281.827} C_DIS
LIN {X 0.104,Y -283.685,Z 1941.562,A 0.000,B 0.000,C 90.000,E1 281.130} C_DIS
LIN {X -0.129,Y -280.859,Z 1941.560,A 0.000,B 0.000,C 90.000,E1 280.838} C_DIS
LIN {X -0.115,Y -274.628,Z 1941.557,A 0.000,B 0.000,C 90.000,E1 280.197} C_DIS
LIN {X -0.037,Y -268.202,Z 1941.553,A 0.000,B 0.000,C 90.000,E1 279.613} C_DIS
LIN {X 0.028,Y -261.551,Z 1941.551,A 0.000,B 0.000,C 90.000,E1 279.095} C_DIS
LIN {X -0.105,Y -254.831,Z 1941.548,A 0.000,B 0.000,C 90.000,E1 278.681} C_DIS
LIN {X -0.039,Y -247.883,Z 1941.546,A 0.000,B 0.000,C 90.000,E1 278.276} C_DIS
LIN {X 0.025,Y -240.396,Z 1941.544,A 0.000,B 0.000,C 90.000,E1 277.936} C_DIS
LIN {X -0.063,Y -232.266,Z 1941.543,A 0.000,B 0.000,C 90.000,E1 277.701} C_DIS
LIN {X 0.086,Y -221.444,Z 1941.542,A 0.000,B 0.000,C 90.000,E1 277.473} C_DIS
LIN {X -0.068,Y -215.364,Z 1941.541,A 0.000,B 0.000,C 90.000,E1 277.466} C_DIS
LIN {X 0.091,Y -180.202,Z 1941.541,A 0.000,B 0.000,C 90.000,E1 277.409} C_DIS
LIN {X 0.029,Y -181.029,Z 1941.530,A 0.000,B 0.000,C 90.000,E1 275.391} C_DIS
LIN {X 0.003,Y -181.579,Z 1941.502,A 0.000,B 0.000,C 90.000,E1 270.344} C_DIS
LIN {X -0.021,Y -180.904,Z 1941.474,A 0.000,B 0.000,C 90.000,E1 265.298} C_DIS
LIN {X -0.071,Y -180.240,Z 1941.464,A 0.000,B 0.000,C 90.000,E1 263.628} C_DIS
LIN {X -0.053,Y -178.727,Z 1941.441,A 0.000,B 0.000,C 90.000,E1 259.398} C_DIS
LIN {X 0.015,Y -175.775,Z 1941.413,A 0.000,B 0.000,C 90.000,E1 254.283} C_DIS
LIN {X 0.003,Y -171.958,Z 1941.384,A 0.000,B 0.000,C 90.000,E1 249.156} C_DIS
LIN {X 0.041,Y -171.352,Z 1941.379,A 0.000,B 0.000,C 90.000,E1 248.284} C_DIS
LIN {X 0.019,Y -167.603,Z 1941.355,A 0.000,B 0.000,C 90.000,E1 243.973} C_DIS
LIN {X 0.031,Y -166.247,Z 1941.346,A 0.000,B 0.000,C 90.000,E1 242.231} C_DIS
LIN {X 0.019,Y -163.003,Z 1941.326,A 0.000,B 0.000,C 90.000,E1 238.742} C_DIS
LIN {X 0.065,Y -160.924,Z 1941.312,A 0.000,B 0.000,C 90.000,E1 236.087} C_DIS
LIN {X 0.042,Y -157.686,Z 1941.292,A 0.000,B 0.000,C 90.000,E1 232.557} C_DIS
LIN {X -0.020,Y -155.725,Z 1941.277,A 0.000,B 0.000,C 90.000,E1 229.908} C_DIS
LIN {X 0.035,Y -151.985,Z 1941.252,A 0.000,B 0.000,C 90.000,E1 225.405} C_DIS
LIN {X 0.051,Y -150.229,Z 1941.237,A 0.000,B 0.000,C 90.000,E1 222.690} C_DIS
LIN {X -0.026,Y -146.990,Z 1941.212,A 0.000,B 0.000,C 90.000,E1 218.177} C_DIS
LIN {X -0.036,Y -145.576,Z 1941.197,A 0.000,B 0.000,C 90.000,E1 215.438} C_DIS
LIN {X 0.081,Y -142.965,Z 1941.171,A 0.000,B 0.000,C 90.000,E1 210.797} C_DIS
LIN {X 0.012,Y -141.592,Z 1941.151,A 0.000,B 0.000,C 90.000,E1 207.129} C_DIS
LIN {X 0.059,Y -139.421,Z 1941.115,A 0.000,B 0.000,C 90.000,E1 200.610} C_DIS
LIN {X -0.021,Y -139.146,Z 1941.104,A 0.000,B 0.000,C 90.000,E1 198.779} C_DIS
LIN {X 0.001,Y -138.346,Z 1941.058,A 0.000,B 0.000,C 90.000,E1 190.366} C_DIS
LIN {X -0.013,Y -139.488,Z 1941.006,A 0.000,B 0.000,C 90.000,E1 181.031} C_DIS
LIN {X 0.067,Y -141.092,Z 1940.975,A 0.000,B 0.000,C 90.000,E1 175.412} C_DIS
LIN {X 0.021,Y -142.470,Z 1940.959,A 0.000,B 0.000,C 90.000,E1 172.648} C_DIS
LIN {X -0.031,Y -144.716,Z 1940.934,A 0.000,B 0.000,C 90.000,E1 168.049} C_DIS
LIN {X 0.062,Y -147.316,Z 1940.913,A 0.000,B 0.000,C 90.000,E1 164.338} C_DIS
LIN {X -0.014,Y -150.637,Z 1940.888,A 0.000,B 0.000,C 90.000,E1 159.806} C_DIS
LIN {X 0.010,Y -154.114,Z 1940.868,A 0.000,B 0.000,C 90.000,E1 156.177} C_DIS
LIN {X -0.066,Y -157.539,Z 1940.848,A 0.000,B 0.000,C 90.000,E1 152.615} C_DIS
LIN {X 0.100,Y -161.776,Z 1940.828,A 0.000,B 0.000,C 90.000,E1 148.997} C_DIS
LIN {X -0.017,Y -165.969,Z 1940.808,A 0.000,B 0.000,C 90.000,E1 145.515} C_DIS
LIN {X -0.021,Y -170.963,Z 1940.789,A 0.000,B 0.000,C 90.000,E1 142.029} C_DIS
LIN {X 0.030,Y -175.832,Z 1940.770,A 0.000,B 0.000,C 90.000,E1 138.566} C_DIS
LIN {X 0.025,Y -181.438,Z 1940.751,A 0.000,B 0.000,C 90.000,E1 135.162} C_DIS
LIN {X -0.101,Y -186.944,Z 1940.732,A 0.000,B 0.000,C 90.000,E1 131.838} C_DIS
LIN {X -0.102,Y -190.057,Z 1940.723,A 0.000,B 0.000,C 90.000,E1 130.172} C_DIS
LIN {X -0.088,Y -195.832,Z 1940.705,A 0.000,B 0.000,C 90.000,E1 126.870} C_DIS
LIN {X -0.020,Y -200.663,Z 1940.691,A 0.000,B 0.000,C 90.000,E1 124.405} C_DIS
LIN {X -0.004,Y -206.549,Z 1940.673,A 0.000,B 0.000,C 90.000,E1 121.180} C_DIS
LIN {X -0.017,Y -209.840,Z 1940.664,A 0.000,B 0.000,C 90.000,E1 119.589} C_DIS
LIN {X 0.002,Y -217.197,Z 1940.642,A 0.000,B 0.000,C 90.000,E1 115.643} C_DIS
LIN {X 0.061,Y -218.824,Z 1940.638,A 0.000,B 0.000,C 90.000,E1 114.847} C_DIS
LIN {X 0.029,Y -224.197,Z 1940.621,A 0.000,B 0.000,C 90.000,E1 111.791} C_DIS
LIN {X 0.110,Y -283.899,Z 1940.621,A 0.000,B 0.000,C 90.000,E1 111.770} C_DIS
LIN {X -0.020,Y -285.537,Z 1940.621,A 0.000,B 0.000,C 90.000,E1 111.770} C_DIS
LIN {X -0.087,Y -288.569,Z 1940.620,A 0.000,B 0.000,C 90.000,E1 111.663} C_DIS
LIN {X -0.050,Y -291.911,Z 1940.619,A 0.000,B 0.000,C 90.000,E1 111.408} C_DIS
LIN {X -0.092,Y -295.573,Z 1940.616,A 0.000,B 0.000,C 90.000,E1 110.972} C_DIS
LIN {X -0.064,Y -312.819,Z 1940.600,A 0.000,B 0.000,C 90.000,E1 108.000} C_DIS
LIN {X 0.110,Y -327.750,Z 1940.587,A 0.000,B 0.000,C 90.000,E1 105.717} C_DIS
LIN {X 0.153,Y -341.754,Z 1940.577,A 0.000,B 0.000,C 90.000,E1 103.828} C_DIS
LIN {X 0.060,Y -356.958,Z 1940.567,A 0.000,B 0.000,C 90.000,E1 102.007} C_DIS
LIN {X 0.032,Y -375.453,Z 1940.556,A 0.000,B 0.000,C 90.000,E1 100.018} C_DIS
LIN {X -0.081,Y -394.412,Z 1940.546,A 0.000,B 0.000,C 90.000,E1 98.219} C_DIS
LIN {X 0.118,Y -416.503,Z 1940.535,A 0.000,B 0.000,C 90.000,E1 96.315} C_DIS
LIN {X -0.046,Y -439.003,Z 1940.526,A 0.000,B 0.000,C 90.000,E1 94.645} C_DIS
LIN {X -0.025,Y -443.229,Z 1940.524,A 0.000,B 0.000,C 90.000,E1 94.245} C_DIS
LIN {X 0.218,Y -446.297,Z 1940.521,A 0.000,B 0.000,C 90.000,E1 93.726} C_DIS
LIN {X 0.133,Y -448.184,Z 1940.518,A 0.000,B 0.000,C 90.000,E1 93.212} C_DIS
LIN {X 0.091,Y -448.993,Z 1940.515,A 0.000,B 0.000,C 90.000,E1 92.694} C_DIS
LIN {X 0.036,Y -448.864,Z 1940.512,A 0.000,B 0.000,C 90.000,E1 92.178} C_DIS
LIN {X 0.004,Y -447.782,Z 1940.509,A 0.000,B 0.000,C 90.000,E1 91.661} C_DIS
LIN {X 0.202,Y -446.838,Z 1940.508,A 0.000,B 0.000,C 90.000,E1 91.375} C_DIS
LIN {X -0.045,Y -445.569,Z 1940.506,A 0.000,B 0.000,C 90.000,E1 91.146} C_DIS
LIN {X -0.103,Y -434.106,Z 1940.496,A 0.000,B 0.000,C 90.000,E1 89.312} C_DIS
LIN {X -0.077,Y -424.092,Z 1940.487,A 0.000,B 0.000,C 90.000,E1 87.707} C_DIS
LIN {X -0.105,Y -412.308,Z 1940.477,A 0.000,B 0.000,C 90.000,E1 85.812} C_DIS
LIN {X -0.028,Y -402.150,Z 1940.467,A 0.000,B 0.000,C 90.000,E1 84.147} C_DIS
LIN {X -0.043,Y -390.164,Z 1940.457,A 0.000,B 0.000,C 90.000,E1 82.186} C_DIS
LIN {X 0.189,Y -378.283,Z 1940.445,A 0.000,B 0.000,C 90.000,E1 80.151} C_DIS
LIN {X 0.147,Y -364.925,Z 1940.432,A 0.000,B 0.000,C 90.000,E1 77.825} C_DIS
LIN {X -0.083,Y -347.602,Z 1940.414,A 0.000,B 0.000,C 90.000,E1 74.574} C_DIS
LIN {X -0.102,Y -334.157,Z 1940.399,A 0.000,B 0.000,C 90.000,E1 71.819} C_DIS
LIN {X 0.184,Y -322.471,Z 1940.385,A 0.000,B 0.000,C 90.000,E1 69.263} C_DIS
LIN {X -0.051,Y -308.503,Z 1940.367,A 0.000,B 0.000,C 90.000,E1 66.102} C_DIS
LIN {X -0.107,Y -300.386,Z 1940.356,A 0.000,B 0.000,C 90.000,E1 64.152} C_DIS
LIN {X 0.044,Y -288.345,Z 1940.340,A 0.000,B 0.000,C 90.000,E1 61.129} C_DIS
LIN {X -0.098,Y -280.284,Z 1940.328,A 0.000,B 0.000,C 90.000,E1 59.125} C_DIS
LIN {X -0.061,Y -270.744,Z 1940.315,A 0.000,B 0.000,C 90.000,E1 56.707} C_DIS
LIN {X -0.073,Y -262.494,Z 1940.303,A 0.000,B 0.000,C 90.000,E1 54.609} C_DIS
LIN {X -0.051,Y -252.889,Z 1940.289,A 0.000,B 0.000,C 90.000,E1 52.110} C_DIS
LIN {X 0.066,Y -243.309,Z 1940.275,A 0.000,B 0.000,C 90.000,E1 49.542} C_DIS
LIN {X 0.046,Y -232.659,Z 1940.259,A 0.000,B 0.000,C 90.000,E1 46.581} C_DIS
LIN {X 0.084,Y -222.384,Z 1940.242,A 0.000,B 0.000,C 90.000,E1 43.542} C_DIS
LIN {X -0.055,Y -211.468,Z 1940.223,A 0.000,B 0.000,C 90.000,E1 40.092} C_DIS
LIN {X -0.023,Y -203.644,Z 1940.207,A 0.000,B 0.000,C 90.000,E1 37.317} C_DIS
LIN {X -0.068,Y -195.517,Z 1940.189,A 0.000,B 0.000,C 90.000,E1 34.119} C_DIS
LIN {X 0.110,Y -188.131,Z 1940.171,A 0.000,B 0.000,C 90.000,E1 30.797} C_DIS
LIN {X -0.019,Y -181.487,Z 1940.153,A 0.000,B 0.000,C 90.000,E1 27.513} C_DIS
LIN {X 0.019,Y -176.961,Z 1940.139,A 0.000,B 0.000,C 90.000,E1 24.975} C_DIS
LIN {X -0.046,Y -171.670,Z 1940.120,A 0.000,B 0.000,C 90.000,E1 21.589} C_DIS
LIN {X -0.009,Y -167.167,Z 1940.101,A 0.000,B 0.000,C 90.000,E1 18.127} C_DIS
LIN {X -0.026,Y -163.524,Z 1940.081,A 0.000,B 0.000,C 90.000,E1 14.647} C_DIS
LIN {X -0.038,Y -159.803,Z 1940.057,A 0.000,B 0.000,C 90.000,E1 10.254} C_DIS
LIN {X 0.022,Y -157.235,Z 1940.032,A 0.000,B 0.000,C 90.000,E1 5.796} C_DIS
LIN {X -0.028,Y -154.928,Z 1939.997,A 0.000,B 0.000,C 90.000,E1 359.542} C_DIS
LIN {X 0.058,Y -154.169,Z 1939.953,A 0.000,B 0.000,C 90.000,E1 351.432} C_DIS
LIN {X -0.019,Y -155.885,Z 1939.913,A 0.000,B 0.000,C 90.000,E1 344.283} C_DIS
LIN {X 0.044,Y -158.593,Z 1939.883,A 0.000,B 0.000,C 90.000,E1 338.901} C_DIS
LIN {X 0.059,Y -162.181,Z 1939.858,A 0.000,B 0.000,C 90.000,E1 334.460} C_DIS
LIN {X -0.034,Y -166.043,Z 1939.839,A 0.000,B 0.000,C 90.000,E1 330.973} C_DIS
LIN {X 0.063,Y -170.904,Z 1939.819,A 0.000,B 0.000,C 90.000,E1 327.454} C_DIS
LIN {X -0.026,Y -175.190,Z 1939.805,A 0.000,B 0.000,C 90.000,E1 324.895} C_DIS
LIN {X 0.027,Y -180.147,Z 1939.791,A 0.000,B 0.000,C 90.000,E1 322.316} C_DIS
LIN {X 0.025,Y -186.003,Z 1939.777,A 0.000,B 0.000,C 90.000,E1 319.784} C_DIS
LIN {X -0.010,Y -191.613,Z 1939.765,A 0.000,B 0.000,C 90.000,E1 317.715} C_DIS
LIN {X 0.026,Y -199.294,Z 1939.751,A 0.000,B 0.000,C 90.000,E1 315.243} C_DIS
LIN {X -0.073,Y -207.882,Z 1939.738,A 0.000,B 0.000,C 90.000,E1 312.852} C_DIS
LIN {X -0.095,Y -218.936,Z 1939.723,A 0.000,B 0.000,C 90.000,E1 310.092} C_DIS
LIN {X -0.031,Y -232.855,Z 1939.705,A 0.000,B 0.000,C 90.000,E1 306.996} C_DIS
LIN {X 0.030,Y -247.911,Z 1939.689,A 0.000,B 0.000,C 90.000,E1 303.992} C_DIS
LIN {X 0.079,Y -259.834,Z 1939.677,A 0.000,B 0.000,C 90.000,E1 301.799} C_DIS
LIN {X 0.082,Y -271.895,Z 1939.665,A 0.000,B 0.000,C 90.000,E1 299.667} C_DIS
LIN {X -0.145,Y -281.798,Z 1939.655,A 0.000,B 0.000,C 90.000,E1 297.975} C_DIS
LIN {X 0.026,Y -291.397,Z 1939.646,A 0.000,B 0.000,C 90.000,E1 296.232} C_DIS
LIN {X 0.106,Y -296.803,Z 1939.640,A 0.000,B 0.000,C 90.000,E1 295.207} C_DIS
LIN {X 0.108,Y -301.601,Z 1939.635,A 0.000,B 0.000,C 90.000,E1 294.207} C_DIS
LIN {X -0.008,Y -304.409,Z 1939.631,A 0.000,B 0.000,C 90.000,E1 293.567} C_DIS
LIN {X 0.053,Y -306.814,Z 1939.627,A 0.000,B 0.000,C 90.000,E1 292.898} C_DIS
LIN {X -0.033,Y -308.823,Z 1939.624,A 0.000,B 0.000,C 90.000,E1 292.259} C_DIS
LIN {X 0.055,Y -310.487,Z 1939.620,A 0.000,B 0.000,C 90.000,E1 291.589} C_DIS
LIN {X -0.133,Y -311.829,Z 1939.616,A 0.000,B 0.000,C 90.000,E1 290.972} C_DIS
LIN {X -0.018,Y -312.824,Z 1939.613,A 0.000,B 0.000,C 90.000,E1 290.301} C_DIS
LIN {X 0.106,Y -313.468,Z 1939.609,A 0.000,B 0.000,C 90.000,E1 289.631} C_DIS
LIN {X -0.163,Y -313.814,Z 1939.606,A 0.000,B 0.000,C 90.000,E1 289.033} C_DIS
LIN {X -0.028,Y -313.803,Z 1939.602,A 0.000,B 0.000,C 90.000,E1 288.362} C_DIS
LIN {X 0.105,Y -313.416,Z 1939.598,A 0.000,B 0.000,C 90.000,E1 287.692} C_DIS
LIN {X 0.145,Y -312.593,Z 1939.595,A 0.000,B 0.000,C 90.000,E1 287.040} C_DIS
LIN {X -0.116,Y -311.283,Z 1939.591,A 0.000,B 0.000,C 90.000,E1 286.441} C_DIS
LIN {X -0.081,Y -309.452,Z 1939.588,A 0.000,B 0.000,C 90.000,E1 285.788} C_DIS
LIN {X -0.055,Y -306.990,Z 1939.584,A 0.000,B 0.000,C 90.000,E1 285.134} C_DIS
LIN {X -0.045,Y -303.756,Z 1939.580,A 0.000,B 0.000,C 90.000,E1 284.481} C_DIS
LIN {X -0.089,Y -296.014,Z 1939.573,A 0.000,B 0.000,C 90.000,E1 283.175} C_DIS
LIN {X 0.073,Y -292.563,Z 1939.569,A 0.000,B 0.000,C 90.000,E1 282.479} C_DIS
LIN {X -0.010,Y -288.576,Z 1939.566,A 0.000,B 0.000,C 90.000,E1 281.827} C_DIS
LIN {X 0.106,Y -283.695,Z 1939.562,A 0.000,B 0.000,C 90.000,E1 281.130} C_DIS
LIN {X -0.125,Y -280.869,Z 1939.560,A 0.000,B 0.000,C 90.000,E1 280.838} C_DIS
LIN {X -0.113,Y -274.629,Z 1939.557,A 0.000,B 0.000,C 90.000,E1 280.197} C_DIS
LIN {X -0.037,Y -268.204,Z 1939.553,A 0.000,B 0.000,C 90.000,E1 279.613} C_DIS
LIN {X 0.029,Y -261.554,Z 1939.551,A 0.000,B 0.000,C 90.000,E1 279.095} C_DIS
LIN {X -0.104,Y -254.829,Z 1939.548,A 0.000,B 0.000,C 90.000,E1 278.681} C_DIS
LIN {X -0.037,Y -247.881,Z 1939.546,A 0.000,B 0.000,C 90.000,E1 278.276} C_DIS
LIN {X 0.027,Y -240.381,Z 1939.544,A 0.000,B 0.000,C 90.000,E1 277.936} C_DIS
LIN {X -0.062,Y -232.253,Z 1939.543,A 0.000,B 0.000,C 90.000,E1 277.701} C_DIS
LIN {X 0.088,Y -221.387,Z 1939.542,A 0.000,B 0.000,C 90.000,E1 277.473} C_DIS
LIN {X -0.066,Y -215.288,Z 1939.541,A 0.000,B 0.000,C 90.000,E1 277.466} C_DIS
LIN {X 0.093,Y -180.203,Z 1939.541,A 0.000,B 0.000,C 90.000,E1 277.409} C_DIS
LIN {X 0.031,Y -181.029,Z 1939.530,A 0.000,B 0.000,C 90.000,E1 275.391} C_DIS
LIN {X 0.006,Y -181.579,Z 1939.502,A 0.000,B 0.000,C 90.000,E1 270.344} C_DIS
LIN {X -0.019,Y -180.903,Z 1939.474,A 0.000,B 0.000,C 90.000,E1 265.298} C_DIS
LIN {X -0.069,Y -180.241,Z 1939.464,A 0.000,B 0.000,C 90.000,E1 263.628} C_DIS
LIN {X -0.049,Y -178.727,Z 1939.441,A 0.000,B 0.000,C 90.000,E1 259.398} C_DIS
LIN {X 0.018,Y -175.775,Z 1939.413,A 0.000,B 0.000,C 90.000,E1 254.283} C_DIS
LIN {X 0.006,Y -171.960,Z 1939.384,A 0.000,B 0.000,C 90.000,E1 249.156} C_DIS
LIN {X 0.042,Y -171.353,Z 1939.379,A 0.000,B 0.000,C 90.000,E1 248.284} C_DIS
LIN {X 0.021,Y -167.603,Z 1939.355,A 0.000,B 0.000,C 90.000,E1 243.973} C_DIS
LIN {X 0.033,Y -166.247,Z 1939.346,A 0.000,B 0.000,C 90.000,E1 242.231} C_DIS
LIN {X 0.021,Y -163.004,Z 1939.326,A 0.000,B 0.000,C 90.000,E1 238.742} C_DIS
LIN {X 0.068,Y -160.925,Z 1939.312,A 0.000,B 0.000,C 90.000,E1 236.087} C_DIS
LIN {X 0.045,Y -157.686,Z 1939.292,A 0.000,B 0.000,C 90.000,E1 232.557} C_DIS
LIN {X -0.017,Y -155.725,Z 1939.277,A 0.000,B 0.000,C 90.000,E1 229.908} C_DIS
LIN {X 0.037,Y -151.985,Z 1939.252,A 0.000,B 0.000,C 90.000,E1 225.405} C_DIS
LIN {X 0.053,Y -150.230,Z 1939.237,A 0.000,B 0.000,C 90.000,E1 222.690} C_DIS
LIN {X -0.024,Y -146.991,Z 1939.212,A 0.000,B 0.000,C 90.000,E1 218.177} C_DIS
LIN {X -0.034,Y -145.576,Z 1939.197,A 0.000,B 0.000,C 90.000,E1 215.438} C_DIS
LIN {X 0.083,Y -142.965,Z 1939.171,A 0.000,B 0.000,C 90.000,E1 210.797} C_DIS
LIN {X 0.013,Y -141.593,Z 1939.151,A 0.000,B 0.000,C 90.000,E1 207.129} C_DIS
LIN {X 0.060,Y -139.420,Z 1939.115,A 0.000,B 0.000,C 90.000,E1 200.610} C_DIS
LIN {X -0.019,Y -139.147,Z 1939.104,A 0.000,B 0.000,C 90.000,E1 198.779} C_DIS
LIN {X 0.003,Y -138.346,Z 1939.058,A 0.000,B 0.000,C 90.000,E1 190.366} C_DIS
LIN {X -0.011,Y -139.488,Z 1939.006,A 0.000,B 0.000,C 90.000,E1 181.031} C_DIS
LIN {X -0.071,Y -141.091,Z 1938.975,A 0.000,B 0.000,C 90.000,E1 175.469} C_DIS
LIN {X 0.023,Y -142.469,Z 1938.959,A 0.000,B 0.000,C 90.000,E1 172.648} C_DIS
LIN {X -0.030,Y -144.716,Z 1938.934,A 0.000,B 0.000,C 90.000,E1 168.049} C_DIS
LIN {X 0.064,Y -147.315,Z 1938.913,A 0.000,B 0.000,C 90.000,E1 164.338} C_DIS
LIN {X -0.064,Y -150.637,Z 1938.888,A 0.000,B 0.000,C 90.000,E1 159.826} C_DIS
LIN {X 0.012,Y -154.113,Z 1938.868,A 0.000,B 0.000,C 90.000,E1 156.177} C_DIS
LIN {X -0.064,Y -157.538,Z 1938.848,A 0.000,B 0.000,C 90.000,E1 152.615} C_DIS
LIN {X 0.101,Y -161.775,Z 1938.828,A 0.000,B 0.000,C 90.000,E1 148.997} C_DIS
LIN {X -0.016,Y -165.968,Z 1938.808,A 0.000,B 0.000,C 90.000,E1 145.515} C_DIS
LIN {X -0.019,Y -170.962,Z 1938.789,A 0.000,B 0.000,C 90.000,E1 142.029} C_DIS
LIN {X 0.032,Y -175.830,Z 1938.770,A 0.000,B 0.000,C 90.000,E1 138.566} C_DIS
LIN {X 0.027,Y -181.437,Z 1938.751,A 0.000,B 0.000,C 90.000,E1 135.162} C_DIS
LIN {X -0.099,Y -186.944,Z 1938.732,A 0.000,B 0.000,C 90.000,E1 131.838} C_DIS
LIN {X -0.100,Y -190.056,Z 1938.723,A 0.000,B 0.000,C 90.000,E1 130.172} C_DIS
LIN {X -0.086,Y -195.831,Z 1938.705,A 0.000,B 0.000,C 90.000,E1 126.870} C_DIS
LIN {X -0.018,Y -200.662,Z 1938.691,A 0.000,B 0.000,C 90.000,E1 124.405} C_DIS
LIN {X -0.002,Y -206.546,Z 1938.673,A 0.000,B 0.000,C 90.000,E1 121.180} C_DIS
LIN {X -0.014,Y -209.838,Z 1938.664,A 0.000,B 0.000,C 90.000,E1 119.589} C_DIS
LIN {X -0.089,Y -217.196,Z 1938.642,A 0.000,B 0.000,C 90.000,E1 115.668} C_DIS
LIN {X 0.063,Y -218.822,Z 1938.638,A 0.000,B 0.000,C 90.000,E1 114.847} C_DIS
LIN {X 0.032,Y -224.196,Z 1938.621,A 0.000,B 0.000,C 90.000,E1 111.791} C_DIS
LIN {X 0.113,Y -283.938,Z 1938.621,A 0.000,B 0.000,C 90.000,E1 111.770} C_DIS
LIN {X -0.017,Y -285.546,Z 1938.621,A 0.000,B 0.000,C 90.000,E1 111.770} C_DIS
LIN {X -0.091,Y -288.596,Z 1938.620,A 0.000,B 0.000,C 90.000,E1 111.663} C_DIS
LIN {X -0.061,Y -291.940,Z 1938.619,A 0.000,B 0.000,C 90.000,E1 111.408} C_DIS
LIN {X -0.115,Y -295.602,Z 1938.616,A 0.000,B 0.000,C 90.000,E1 110.972} C_DIS
LIN {X -0.100,Y -312.858,Z 1938.600,A 0.000,B 0.000,C 90.000,E1 108.000} C_DIS
LIN {X 0.074,Y -327.793,Z 1938.587,A 0.000,B 0.000,C 90.000,E1 105.717} C_DIS
LIN {X 0.115,Y -341.801,Z 1938.577,A 0.000,B 0.000,C 90.000,E1 103.828} C_DIS
LIN {X 0.023,Y -357.008,Z 1938.567,A 0.000,B 0.000,C 90.000,E1 102.007} C_DIS
LIN {X -0.003,Y -375.505,Z 1938.556,A 0.000,B 0.000,C 90.000,E1 100.018} C_DIS
LIN {X -0.115,Y -394.464,Z 1938.546,A 0.000,B 0.000,C 90.000,E1 98.219} C_DIS
LIN {X 0.086,Y -416.557,Z 1938.535,A 0.000,B 0.000,C 90.000,E1 96.315} C_DIS
LIN {X -0.077,Y -439.058,Z 1938.526,A 0.000,B 0.000,C 90.000,E1 94.645} C_DIS
LIN {X -0.056,Y -443.254,Z 1938.524,A 0.000,B 0.000,C 90.000,E1 94.245} C_DIS
LIN {X 0.170,Y -446.316,Z 1938.521,A 0.000,B 0.000,C 90.000,E1 93.726} C_DIS
LIN {X 0.085,Y -448.187,Z 1938.518,A 0.000,B 0.000,C 90.000,E1 93.212} C_DIS
LIN {X 0.042,Y -448.983,Z 1938.515,A 0.000,B 0.000,C 90.000,E1 92.694} C_DIS
LIN {X -0.012,Y -448.841,Z 1938.512,A 0.000,B 0.000,C 90.000,E1 92.178} C_DIS
LIN {X -0.044,Y -447.746,Z 1938.509,A 0.000,B 0.000,C 90.000,E1 91.661} C_DIS
LIN {X 0.154,Y -446.794,Z 1938.508,A 0.000,B 0.000,C 90.000,E1 91.375} C_DIS
LIN {X -0.093,Y -445.515,Z 1938.506,A 0.000,B 0.000,C 90.000,E1 91.146} C_DIS
LIN {X -0.151,Y -434.048,Z 1938.496,A 0.000,B 0.000,C 90.000,E1 89.312} C_DIS
LIN {X -0.124,Y -424.030,Z 1938.487,A 0.000,B 0.000,C 90.000,E1 87.707} C_DIS
LIN {X -0.152,Y -412.250,Z 1938.477,A 0.000,B 0.000,C 90.000,E1 85.812} C_DIS
LIN {X -0.075,Y -402.092,Z 1938.467,A 0.000,B 0.000,C 90.000,E1 84.147} C_DIS
LIN {X -0.091,Y -390.105,Z 1938.457,A 0.000,B 0.000,C 90.000,E1 82.186} C_DIS
LIN {X 0.142,Y -378.224,Z 1938.445,A 0.000,B 0.000,C 90.000,E1 80.151} C_DIS
LIN {X 0.157,Y -363.236,Z 1938.431,A 0.000,B 0.000,C 90.000,E1 77.521} C_DIS
LIN {X -0.107,Y -346.032,Z 1938.412,A 0.000,B 0.000,C 90.000,E1 74.267} C_DIS
LIN {X -0.149,Y -334.099,Z 1938.399,A 0.000,B 0.000,C 90.000,E1 71.819} C_DIS
LIN {X 0.178,Y -323.851,Z 1938.387,A 0.000,B 0.000,C 90.000,E1 69.571} C_DIS
LIN {X -0.016,Y -309.793,Z 1938.369,A 0.000,B 0.000,C 90.000,E1 66.410} C_DIS
LIN {X -0.152,Y -300.328,Z 1938.356,A 0.000,B 0.000,C 90.000,E1 64.152} C_DIS
LIN {X -0.002,Y -288.287,Z 1938.340,A 0.000,B 0.000,C 90.000,E1 61.129} C_DIS
LIN {X 0.098,Y -280.225,Z 1938.328,A 0.000,B 0.000,C 90.000,E1 59.076} C_DIS
LIN {X -0.105,Y -270.687,Z 1938.315,A 0.000,B 0.000,C 90.000,E1 56.707} C_DIS
LIN {X 0.097,Y -262.437,Z 1938.303,A 0.000,B 0.000,C 90.000,E1 54.562} C_DIS
LIN {X -0.095,Y -252.834,Z 1938.289,A 0.000,B 0.000,C 90.000,E1 52.110} C_DIS
LIN {X 0.023,Y -243.254,Z 1938.275,A 0.000,B 0.000,C 90.000,E1 49.542} C_DIS
LIN {X 0.003,Y -232.605,Z 1938.259,A 0.000,B 0.000,C 90.000,E1 46.581} C_DIS
LIN {X 0.041,Y -222.331,Z 1938.242,A 0.000,B 0.000,C 90.000,E1 43.542} C_DIS
LIN {X -0.097,Y -211.417,Z 1938.223,A 0.000,B 0.000,C 90.000,E1 40.092} C_DIS
LIN {X -0.064,Y -203.601,Z 1938.207,A 0.000,B 0.000,C 90.000,E1 37.317} C_DIS
LIN {X 0.053,Y -195.477,Z 1938.189,A 0.000,B 0.000,C 90.000,E1 34.072} C_DIS
LIN {X 0.069,Y -188.095,Z 1938.171,A 0.000,B 0.000,C 90.000,E1 30.797} C_DIS
LIN {X -0.058,Y -181.456,Z 1938.153,A 0.000,B 0.000,C 90.000,E1 27.513} C_DIS
LIN {X 0.055,Y -176.933,Z 1938.139,A 0.000,B 0.000,C 90.000,E1 24.951} C_DIS
LIN {X 0.076,Y -171.645,Z 1938.120,A 0.000,B 0.000,C 90.000,E1 21.535} C_DIS
LIN {X -0.047,Y -167.146,Z 1938.101,A 0.000,B 0.000,C 90.000,E1 18.127} C_DIS
LIN {X 0.094,Y -163.504,Z 1938.081,A 0.000,B 0.000,C 90.000,E1 14.592} C_DIS
LIN {X -0.076,Y -159.786,Z 1938.057,A 0.000,B 0.000,C 90.000,E1 10.254} C_DIS
LIN {X -0.015,Y -157.219,Z 1938.032,A 0.000,B 0.000,C 90.000,E1 5.796} C_DIS
LIN {X -0.028,Y -154.919,Z 1937.997,A 0.000,B 0.000,C 90.000,E1 359.542} C_DIS
LIN {X 0.058,Y -154.161,Z 1937.953,A 0.000,B 0.000,C 90.000,E1 351.432} C_DIS
LIN {X -0.021,Y -155.879,Z 1937.913,A 0.000,B 0.000,C 90.000,E1 344.283} C_DIS
LIN {X 0.043,Y -158.590,Z 1937.883,A 0.000,B 0.000,C 90.000,E1 338.901} C_DIS
LIN {X 0.058,Y -162.179,Z 1937.858,A 0.000,B 0.000,C 90.000,E1 334.460} C_DIS
LIN {X -0.036,Y -166.045,Z 1937.839,A 0.000,B 0.000,C 90.000,E1 330.973} C_DIS
LIN {X 0.062,Y -170.908,Z 1937.819,A 0.000,B 0.000,C 90.000,E1 327.454} C_DIS
LIN {X -0.027,Y -175.197,Z 1937.805,A 0.000,B 0.000,C 90.000,E1 324.895} C_DIS
LIN {X 0.025,Y -180.156,Z 1937.791,A 0.000,B 0.000,C 90.000,E1 322.316} C_DIS
LIN {X 0.024,Y -186.012,Z 1937.777,A 0.000,B 0.000,C 90.000,E1 319.784} C_DIS
LIN {X -0.011,Y -191.623,Z 1937.765,A 0.000,B 0.000,C 90.000,E1 317.715} C_DIS
LIN {X 0.025,Y -199.300,Z 1937.751,A 0.000,B 0.000,C 90.000,E1 315.243} C_DIS
LIN {X -0.074,Y -207.888,Z 1937.738,A 0.000,B 0.000,C 90.000,E1 312.852} C_DIS
LIN {X -0.095,Y -218.944,Z 1937.723,A 0.000,B 0.000,C 90.000,E1 310.092} C_DIS
LIN {X -0.031,Y -232.864,Z 1937.705,A 0.000,B 0.000,C 90.000,E1 306.996} C_DIS
LIN {X 0.030,Y -247.921,Z 1937.689,A 0.000,B 0.000,C 90.000,E1 303.992} C_DIS
LIN {X 0.079,Y -259.845,Z 1937.677,A 0.000,B 0.000,C 90.000,E1 301.799} C_DIS
LIN {X 0.083,Y -271.906,Z 1937.665,A 0.000,B 0.000,C 90.000,E1 299.667} C_DIS
LIN {X -0.144,Y -281.806,Z 1937.655,A 0.000,B 0.000,C 90.000,E1 297.975} C_DIS
LIN {X 0.027,Y -291.406,Z 1937.646,A 0.000,B 0.000,C 90.000,E1 296.232} C_DIS
LIN {X 0.107,Y -296.814,Z 1937.640,A 0.000,B 0.000,C 90.000,E1 295.207} C_DIS
LIN {X 0.108,Y -301.614,Z 1937.635,A 0.000,B 0.000,C 90.000,E1 294.207} C_DIS
LIN {X -0.006,Y -304.422,Z 1937.631,A 0.000,B 0.000,C 90.000,E1 293.567} C_DIS
LIN {X 0.054,Y -306.826,Z 1937.627,A 0.000,B 0.000,C 90.000,E1 292.898} C_DIS
LIN {X -0.032,Y -308.836,Z 1937.624,A 0.000,B 0.000,C 90.000,E1 292.259} C_DIS
LIN {X 0.056,Y -310.501,Z 1937.620,A 0.000,B 0.000,C 90.000,E1 291.589} C_DIS
LIN {X -0.131,Y -311.844,Z 1937.616,A 0.000,B 0.000,C 90.000,E1 290.972} C_DIS
LIN {X -0.017,Y -312.839,Z 1937.613,A 0.000,B 0.000,C 90.000,E1 290.301} C_DIS
LIN {X 0.107,Y -313.484,Z 1937.609,A 0.000,B 0.000,C 90.000,E1 289.631} C_DIS
LIN {X -0.162,Y -313.828,Z 1937.606,A 0.000,B 0.000,C 90.000,E1 289.033} C_DIS
LIN {X -0.027,Y -313.818,Z 1937.602,A 0.000,B 0.000,C 90.000,E1 288.362} C_DIS
LIN {X 0.108,Y -313.430,Z 1937.598,A 0.000,B 0.000,C 90.000,E1 287.692} C_DIS
LIN {X 0.147,Y -312.611,Z 1937.595,A 0.000,B 0.000,C 90.000,E1 287.040} C_DIS
LIN {X -0.114,Y -311.303,Z 1937.591,A 0.000,B 0.000,C 90.000,E1 286.441} C_DIS
LIN {X -0.079,Y -309.468,Z 1937.588,A 0.000,B 0.000,C 90.000,E1 285.788} C_DIS
LIN {X -0.052,Y -307.009,Z 1937.584,A 0.000,B 0.000,C 90.000,E1 285.134} C_DIS
LIN {X -0.043,Y -303.774,Z 1937.580,A 0.000,B 0.000,C 90.000,E1 284.481} C_DIS
LIN {X -0.087,Y -296.035,Z 1937.573,A 0.000,B 0.000,C 90.000,E1 283.175} C_DIS
LIN {X 0.075,Y -292.577,Z 1937.569,A 0.000,B 0.000,C 90.000,E1 282.479} C_DIS
LIN {X -0.008,Y -288.589,Z 1937.566,A 0.000,B 0.000,C 90.000,E1 281.827} C_DIS
LIN {X 0.109,Y -283.704,Z 1937.562,A 0.000,B 0.000,C 90.000,E1 281.130} C_DIS
LIN {X -0.123,Y -280.879,Z 1937.560,A 0.000,B 0.000,C 90.000,E1 280.838} C_DIS
LIN {X -0.111,Y -274.631,Z 1937.557,A 0.000,B 0.000,C 90.000,E1 280.197} C_DIS
LIN {X -0.036,Y -268.206,Z 1937.553,A 0.000,B 0.000,C 90.000,E1 279.613} C_DIS
LIN {X 0.029,Y -261.557,Z 1937.551,A 0.000,B 0.000,C 90.000,E1 279.095} C_DIS
LIN {X -0.102,Y -254.830,Z 1937.548,A 0.000,B 0.000,C 90.000,E1 278.681} C_DIS
LIN {X -0.035,Y -247.882,Z 1937.546,A 0.000,B 0.000,C 90.000,E1 278.276} C_DIS
LIN {X 0.029,Y -240.374,Z 1937.544,A 0.000,B 0.000,C 90.000,E1 277.936} C_DIS
LIN {X -0.060,Y -232.254,Z 1937.543,A 0.000,B 0.000,C 90.000,E1 277.701} C_DIS
LIN {X 0.090,Y -221.359,Z 1937.542,A 0.000,B 0.000,C 90.000,E1 277.473} C_DIS
LIN {X -0.063,Y -215.254,Z 1937.541,A 0.000,B 0.000,C 90.000,E1 277.466} C_DIS
LIN {X 0.096,Y -180.202,Z 1937.541,A 0.000,B 0.000,C 90.000,E1 277.409} C_DIS
LIN {X 0.034,Y -181.029,Z 1937.530,A 0.000,B 0.000,C 90.000,E1 275.391} C_DIS
LIN {X 0.009,Y -181.579,Z 1937.502,A 0.000,B 0.000,C 90.000,E1 270.344} C_DIS
LIN {X -0.016,Y -180.903,Z 1937.474,A 0.000,B 0.000,C 90.000,E1 265.298} C_DIS
LIN {X -0.066,Y -180.241,Z 1937.464,A 0.000,B 0.000,C 90.000,E1 263.628} C_DIS
LIN {X -0.047,Y -178.728,Z 1937.441,A 0.000,B 0.000,C 90.000,E1 259.398} C_DIS
LIN {X 0.021,Y -175.776,Z 1937.413,A 0.000,B 0.000,C 90.000,E1 254.283} C_DIS
LIN {X 0.009,Y -171.959,Z 1937.384,A 0.000,B 0.000,C 90.000,E1 249.156} C_DIS
LIN {X 0.046,Y -171.353,Z 1937.379,A 0.000,B 0.000,C 90.000,E1 248.284} C_DIS
LIN {X 0.024,Y -167.604,Z 1937.355,A 0.000,B 0.000,C 90.000,E1 243.973} C_DIS
LIN {X 0.036,Y -166.249,Z 1937.346,A 0.000,B 0.000,C 90.000,E1 242.231} C_DIS
LIN {X 0.023,Y -163.004,Z 1937.326,A 0.000,B 0.000,C 90.000,E1 238.742} C_DIS
LIN {X 0.070,Y -160.926,Z 1937.312,A 0.000,B 0.000,C 90.000,E1 236.087} C_DIS
LIN {X 0.047,Y -157.687,Z 1937.292,A 0.000,B 0.000,C 90.000,E1 232.557} C_DIS
LIN {X -0.014,Y -155.727,Z 1937.277,A 0.000,B 0.000,C 90.000,E1 229.908} C_DIS
LIN {X 0.039,Y -151.986,Z 1937.252,A 0.000,B 0.000,C 90.000,E1 225.405} C_DIS
LIN {X 0.055,Y -150.230,Z 1937.237,A 0.000,B 0.000,C 90.000,E1 222.690} C_DIS
LIN {X -0.021,Y -146.992,Z 1937.212,A 0.000,B 0.000,C 90.000,E1 218.177} C_DIS
LIN {X -0.031,Y -145.577,Z 1937.197,A 0.000,B 0.000,C 90.000,E1 215.438} C_DIS
LIN {X -0.037,Y -142.967,Z 1937.171,A 0.000,B 0.000,C 90.000,E1 210.846} C_DIS
LIN {X 0.017,Y -141.593,Z 1937.151,A 0.000,B 0.000,C 90.000,E1 207.129} C_DIS
LIN {X 0.063,Y -139.420,Z 1937.115,A 0.000,B 0.000,C 90.000,E1 200.610} C_DIS
LIN {X -0.016,Y -139.147,Z 1937.104,A 0.000,B 0.000,C 90.000,E1 198.779} C_DIS
LIN {X 0.006,Y -138.346,Z 1937.058,A 0.000,B 0.000,C 90.000,E1 190.366} C_DIS
LIN {X -0.009,Y -139.487,Z 1937.006,A 0.000,B 0.000,C 90.000,E1 181.031} C_DIS
LIN {X -0.068,Y -141.091,Z 1936.975,A 0.000,B 0.000,C 90.000,E1 175.469} C_DIS
LIN {X 0.025,Y -142.469,Z 1936.959,A 0.000,B 0.000,C 90.000,E1 172.648} C_DIS
LIN {X -0.027,Y -144.715,Z 1936.934,A 0.000,B 0.000,C 90.000,E1 168.049} C_DIS
LIN {X 0.067,Y -147.315,Z 1936.913,A 0.000,B 0.000,C 90.000,E1 164.338} C_DIS
LIN {X -0.061,Y -150.635,Z 1936.888,A 0.000,B 0.000,C 90.000,E1 159.826} C_DIS
LIN {X 0.015,Y -154.113,Z 1936.868,A 0.000,B 0.000,C 90.000,E1 156.177} C_DIS
LIN {X -0.061,Y -157.536,Z 1936.848,A 0.000,B 0.000,C 90.000,E1 152.615} C_DIS
LIN {X 0.104,Y -161.774,Z 1936.828,A 0.000,B 0.000,C 90.000,E1 148.997} C_DIS
LIN {X -0.012,Y -165.966,Z 1936.808,A 0.000,B 0.000,C 90.000,E1 145.515} C_DIS
LIN {X -0.016,Y -170.960,Z 1936.789,A 0.000,B 0.000,C 90.000,E1 142.029} C_DIS
LIN {X 0.035,Y -175.829,Z 1936.770,A 0.000,B 0.000,C 90.000,E1 138.566} C_DIS
LIN {X 0.031,Y -181.435,Z 1936.751,A 0.000,B 0.000,C 90.000,E1 135.162} C_DIS
LIN {X -0.096,Y -186.941,Z 1936.732,A 0.000,B 0.000,C 90.000,E1 131.838} C_DIS
LIN {X -0.097,Y -190.054,Z 1936.723,A 0.000,B 0.000,C 90.000,E1 130.172} C_DIS
LIN {X -0.082,Y -195.829,Z 1936.705,A 0.000,B 0.000,C 90.000,E1 126.870} C_DIS
LIN {X -0.015,Y -200.661,Z 1936.691,A 0.000,B 0.000,C 90.000,E1 124.405} C_DIS
LIN {X 0.002,Y -206.545,Z 1936.673,A 0.000,B 0.000,C 90.000,E1 121.180} C_DIS
LIN {X -0.011,Y -209.837,Z 1936.664,A 0.000,B 0.000,C 90.000,E1 119.589} C_DIS
LIN {X -0.086,Y -217.194,Z 1936.642,A 0.000,B 0.000,C 90.000,E1 115.668} C_DIS
LIN {X 0.067,Y -218.821,Z 1936.638,A 0.000,B 0.000,C 90.000,E1 114.847} C_DIS
LIN {X 0.036,Y -224.194,Z 1936.621,A 0.000,B 0.000,C 90.000,E1 111.791} C_DIS
LIN {X 0.117,Y -283.949,Z 1936.621,A 0.000,B 0.000,C 90.000,E1 111.770} C_DIS
LIN {X -0.012,Y -285.546,Z 1936.621,A 0.000,B 0.000,C 90.000,E1 111.770} C_DIS
LIN {X -0.089,Y -288.602,Z 1936.620,A 0.000,B 0.000,C 90.000,E1 111.663} C_DIS
LIN {X -0.063,Y -291.947,Z 1936.619,A 0.000,B 0.000,C 90.000,E1 111.408} C_DIS
LIN {X -0.120,Y -295.609,Z 1936.616,A 0.000,B 0.000,C 90.000,E1 110.972} C_DIS
LIN {X -0.110,Y -312.869,Z 1936.600,A 0.000,B 0.000,C 90.000,E1 108.000} C_DIS
LIN {X 0.063,Y -327.806,Z 1936.587,A 0.000,B 0.000,C 90.000,E1 105.717} C_DIS
LIN {X 0.105,Y -341.813,Z 1936.577,A 0.000,B 0.000,C 90.000,E1 103.828} C_DIS
LIN {X 0.011,Y -357.022,Z 1936.567,A 0.000,B 0.000,C 90.000,E1 102.007} C_DIS
LIN {X -0.014,Y -375.519,Z 1936.556,A 0.000,B 0.000,C 90.000,E1 100.018} C_DIS
LIN {X -0.125,Y -394.479,Z 1936.546,A 0.000,B 0.000,C 90.000,E1 98.219} C_DIS
LIN {X 0.077,Y -416.572,Z 1936.535,A 0.000,B 0.000,C 90.000,E1 96.315} C_DIS
LIN {X -0.086,Y -439.072,Z 1936.526,A 0.000,B 0.000,C 90.000,E1 94.645} C_DIS
LIN {X -0.078,Y -443.268,Z 1936.524,A 0.000,B 0.000,C 90.000,E1 94.245} C_DIS
LIN {X 0.139,Y -446.325,Z 1936.521,A 0.000,B 0.000,C 90.000,E1 93.726} C_DIS
LIN {X 0.053,Y -448.184,Z 1936.518,A 0.000,B 0.000,C 90.000,E1 93.212} C_DIS
LIN {X 0.011,Y -448.971,Z 1936.515,A 0.000,B 0.000,C 90.000,E1 92.694} C_DIS
LIN {X -0.043,Y -448.821,Z 1936.512,A 0.000,B 0.000,C 90.000,E1 92.178} C_DIS
LIN {X -0.076,Y -447.716,Z 1936.509,A 0.000,B 0.000,C 90.000,E1 91.661} C_DIS
LIN {X 0.123,Y -446.759,Z 1936.508,A 0.000,B 0.000,C 90.000,E1 91.375} C_DIS
LIN {X -0.125,Y -445.473,Z 1936.506,A 0.000,B 0.000,C 90.000,E1 91.146} C_DIS
LIN {X -0.182,Y -434.003,Z 1936.496,A 0.000,B 0.000,C 90.000,E1 89.312} C_DIS
LIN {X -0.156,Y -423.984,Z 1936.487,A 0.000,B 0.000,C 90.000,E1 87.707} C_DIS
LIN {X -0.185,Y -412.204,Z 1936.477,A 0.000,B 0.000,C 90.000,E1 85.812} C_DIS
LIN {X -0.108,Y -402.046,Z 1936.467,A 0.000,B 0.000,C 90.000,E1 84.147} C_DIS
LIN {X -0.123,Y -390.060,Z 1936.457,A 0.000,B 0.000,C 90.000,E1 82.186} C_DIS
LIN {X 0.110,Y -378.177,Z 1936.445,A 0.000,B 0.000,C 90.000,E1 80.151} C_DIS
LIN {X 0.125,Y -363.187,Z 1936.431,A 0.000,B 0.000,C 90.000,E1 77.521} C_DIS
LIN {X 0.194,Y -345.987,Z 1936.412,A 0.000,B 0.000,C 90.000,E1 74.212} C_DIS
LIN {X 0.137,Y -334.053,Z 1936.399,A 0.000,B 0.000,C 90.000,E1 71.764} C_DIS
LIN {X 0.146,Y -323.806,Z 1936.387,A 0.000,B 0.000,C 90.000,E1 69.571} C_DIS
LIN {X -0.048,Y -309.748,Z 1936.369,A 0.000,B 0.000,C 90.000,E1 66.410} C_DIS
LIN {X 0.087,Y -300.280,Z 1936.356,A 0.000,B 0.000,C 90.000,E1 64.101} C_DIS
LIN {X -0.034,Y -288.240,Z 1936.340,A 0.000,B 0.000,C 90.000,E1 61.129} C_DIS
LIN {X 0.066,Y -280.178,Z 1936.328,A 0.000,B 0.000,C 90.000,E1 59.076} C_DIS
LIN {X -0.137,Y -270.641,Z 1936.315,A 0.000,B 0.000,C 90.000,E1 56.707} C_DIS
LIN {X 0.152,Y -263.792,Z 1936.305,A 0.000,B 0.000,C 90.000,E1 54.895} C_DIS
LIN {X 0.072,Y -252.792,Z 1936.289,A 0.000,B 0.000,C 90.000,E1 52.065} C_DIS
LIN {X -0.009,Y -243.210,Z 1936.275,A 0.000,B 0.000,C 90.000,E1 49.542} C_DIS
LIN {X -0.028,Y -232.561,Z 1936.259,A 0.000,B 0.000,C 90.000,E1 46.581} C_DIS
LIN {X 0.010,Y -222.286,Z 1936.242,A 0.000,B 0.000,C 90.000,E1 43.542} C_DIS
LIN {X -0.126,Y -211.376,Z 1936.223,A 0.000,B 0.000,C 90.000,E1 40.092} C_DIS
LIN {X 0.030,Y -203.564,Z 1936.207,A 0.000,B 0.000,C 90.000,E1 37.282} C_DIS
LIN {X 0.024,Y -195.444,Z 1936.189,A 0.000,B 0.000,C 90.000,E1 34.072} C_DIS
LIN {X 0.040,Y -188.067,Z 1936.171,A 0.000,B 0.000,C 90.000,E1 30.797} C_DIS
LIN {X -0.088,Y -181.430,Z 1936.153,A 0.000,B 0.000,C 90.000,E1 27.513} C_DIS
LIN {X 0.026,Y -176.909,Z 1936.139,A 0.000,B 0.000,C 90.000,E1 24.951} C_DIS
LIN {X 0.047,Y -171.625,Z 1936.120,A 0.000,B 0.000,C 90.000,E1 21.535} C_DIS
LIN {X -0.023,Y -167.128,Z 1936.101,A 0.000,B 0.000,C 90.000,E1 18.109} C_DIS
LIN {X 0.066,Y -163.487,Z 1936.081,A 0.000,B 0.000,C 90.000,E1 14.592} C_DIS
LIN {X 0.053,Y -159.771,Z 1936.057,A 0.000,B 0.000,C 90.000,E1 10.197} C_DIS
LIN {X -0.043,Y -157.205,Z 1936.032,A 0.000,B 0.000,C 90.000,E1 5.796} C_DIS
LIN {X -0.028,Y -154.910,Z 1935.997,A 0.000,B 0.000,C 90.000,E1 359.542} C_DIS
LIN {X 0.058,Y -154.154,Z 1935.953,A 0.000,B 0.000,C 90.000,E1 351.432} C_DIS
LIN {X -0.021,Y -155.874,Z 1935.913,A 0.000,B 0.000,C 90.000,E1 344.283} C_DIS
LIN {X 0.041,Y -158.586,Z 1935.883,A 0.000,B 0.000,C 90.000,E1 338.901} C_DIS
LIN {X 0.057,Y -162.177,Z 1935.858,A 0.000,B 0.000,C 90.000,E1 334.460} C_DIS
LIN {X -0.037,Y -166.046,Z 1935.839,A 0.000,B 0.000,C 90.000,E1 330.973} C_DIS
LIN {X 0.061,Y -170.913,Z 1935.819,A 0.000,B 0.000,C 90.000,E1 327.454} C_DIS
LIN {X -0.028,Y -175.204,Z 1935.805,A 0.000,B 0.000,C 90.000,E1 324.895} C_DIS
LIN {X 0.024,Y -180.164,Z 1935.791,A 0.000,B 0.000,C 90.000,E1 322.316} C_DIS
LIN {X 0.023,Y -186.021,Z 1935.777,A 0.000,B 0.000,C 90.000,E1 319.784} C_DIS
LIN {X -0.012,Y -191.632,Z 1935.765,A 0.000,B 0.000,C 90.000,E1 317.715} C_DIS
LIN {X 0.025,Y -199.306,Z 1935.751,A 0.000,B 0.000,C 90.000,E1 315.243} C_DIS
LIN {X -0.074,Y -207.895,Z 1935.738,A 0.000,B 0.000,C 90.000,E1 312.852} C_DIS
LIN {X -0.095,Y -218.952,Z 1935.723,A 0.000,B 0.000,C 90.000,E1 310.092} C_DIS
LIN {X -0.031,Y -232.874,Z 1935.705,A 0.000,B 0.000,C 90.000,E1 306.996} C_DIS
LIN {X 0.030,Y -247.932,Z 1935.689,A 0.000,B 0.000,C 90.000,E1 303.992} C_DIS
LIN {X 0.080,Y -259.856,Z 1935.677,A 0.000,B 0.000,C 90.000,E1 301.799} C_DIS
LIN {X 0.084,Y -271.917,Z 1935.665,A 0.000,B 0.000,C 90.000,E1 299.667} C_DIS
LIN {X -0.143,Y -281.816,Z 1935.655,A 0.000,B 0.000,C 90.000,E1 297.975} C_DIS
LIN {X 0.028,Y -291.416,Z 1935.646,A 0.000,B 0.000,C 90.000,E1 296.232} C_DIS
LIN {X 0.108,Y -296.826,Z 1935.640,A 0.000,B 0.000,C 90.000,E1 295.207} C_DIS
LIN {X 0.109,Y -301.626,Z 1935.635,A 0.000,B 0.000,C 90.000,E1 294.207} C_DIS
LIN {X -0.005,Y -304.435,Z 1935.631,A 0.000,B 0.000,C 90.000,E1 293.567} C_DIS
LIN {X 0.055,Y -306.838,Z 1935.627,A 0.000,B 0.000,C 90.000,E1 292.898} C_DIS
LIN {X -0.031,Y -308.849,Z 1935.624,A 0.000,B 0.000,C 90.000,E1 292.259} C_DIS
LIN {X 0.058,Y -310.516,Z 1935.620,A 0.000,B 0.000,C 90.000,E1 291.589} C_DIS
LIN {X -0.129,Y -311.859,Z 1935.616,A 0.000,B 0.000,C 90.000,E1 290.972} C_DIS
LIN {X -0.015,Y -312.856,Z 1935.613,A 0.000,B 0.000,C 90.000,E1 290.301} C_DIS
LIN {X 0.109,Y -313.498,Z 1935.609,A 0.000,B 0.000,C 90.000,E1 289.631} C_DIS
LIN {X -0.160,Y -313.842,Z 1935.606,A 0.000,B 0.000,C 90.000,E1 289.033} C_DIS
LIN {X -0.025,Y -313.833,Z 1935.602,A 0.000,B 0.000,C 90.000,E1 288.362} C_DIS
LIN {X 0.110,Y -313.446,Z 1935.598,A 0.000,B 0.000,C 90.000,E1 287.692} C_DIS
LIN {X 0.149,Y -312.628,Z 1935.595,A 0.000,B 0.000,C 90.000,E1 287.040} C_DIS
LIN {X -0.112,Y -311.322,Z 1935.591,A 0.000,B 0.000,C 90.000,E1 286.441} C_DIS
LIN {X -0.077,Y -309.485,Z 1935.588,A 0.000,B 0.000,C 90.000,E1 285.788} C_DIS
LIN {X -0.050,Y -307.028,Z 1935.584,A 0.000,B 0.000,C 90.000,E1 285.134} C_DIS
LIN {X -0.041,Y -303.792,Z 1935.580,A 0.000,B 0.000,C 90.000,E1 284.481} C_DIS
LIN {X -0.085,Y -296.055,Z 1935.573,A 0.000,B 0.000,C 90.000,E1 283.175} C_DIS
LIN {X 0.001,Y -290.820,Z 1935.568,A 0.000,B 0.000,C 90.000,E1 282.187} C_DIS
LIN {X -0.092,Y -286.457,Z 1935.564,A 0.000,B 0.000,C 90.000,E1 281.535} C_DIS
LIN {X 0.014,Y -281.122,Z 1935.560,A 0.000,B 0.000,C 90.000,E1 280.838} C_DIS
LIN {X 0.012,Y -274.900,Z 1935.557,A 0.000,B 0.000,C 90.000,E1 280.197} C_DIS
LIN {X 0.066,Y -268.457,Z 1935.553,A 0.000,B 0.000,C 90.000,E1 279.613} C_DIS
LIN {X 0.113,Y -261.813,Z 1935.551,A 0.000,B 0.000,C 90.000,E1 279.095} C_DIS
LIN {X -0.036,Y -255.080,Z 1935.548,A 0.000,B 0.000,C 90.000,E1 278.681} C_DIS
LIN {X 0.024,Y -248.135,Z 1935.546,A 0.000,B 0.000,C 90.000,E1 278.276} C_DIS
LIN {X 0.079,Y -240.658,Z 1935.544,A 0.000,B 0.000,C 90.000,E1 277.936} C_DIS
LIN {X -0.022,Y -232.599,Z 1935.543,A 0.000,B 0.000,C 90.000,E1 277.701} C_DIS
LIN {X -0.101,Y -221.943,Z 1935.542,A 0.000,B 0.000,C 90.000,E1 277.530} C_DIS
LIN {X -0.037,Y -216.135,Z 1935.541,A 0.000,B 0.000,C 90.000,E1 277.466} C_DIS
LIN {X -0.062,Y -180.200,Z 1935.541,A 0.000,B 0.000,C 90.000,E1 277.466} C_DIS
LIN {X 0.054,Y -181.028,Z 1935.530,A 0.000,B 0.000,C 90.000,E1 275.391} C_DIS
LIN {X 0.029,Y -181.578,Z 1935.502,A 0.000,B 0.000,C 90.000,E1 270.344} C_DIS
LIN {X 0.004,Y -180.903,Z 1935.474,A 0.000,B 0.000,C 90.000,E1 265.298} C_DIS
LIN {X -0.046,Y -180.245,Z 1935.464,A 0.000,B 0.000,C 90.000,E1 263.628} C_DIS
LIN {X -0.027,Y -178.732,Z 1935.441,A 0.000,B 0.000,C 90.000,E1 259.398} C_DIS
LIN {X 0.040,Y -175.779,Z 1935.413,A 0.000,B 0.000,C 90.000,E1 254.283} C_DIS
LIN {X 0.029,Y -171.964,Z 1935.384,A 0.000,B 0.000,C 90.000,E1 249.156} C_DIS
LIN {X 0.066,Y -171.360,Z 1935.380,A 0.000,B 0.000,C 90.000,E1 248.284} C_DIS
LIN {X 0.043,Y -167.609,Z 1935.355,A 0.000,B 0.000,C 90.000,E1 243.973} C_DIS
LIN {X 0.055,Y -166.256,Z 1935.346,A 0.000,B 0.000,C 90.000,E1 242.231} C_DIS
LIN {X 0.043,Y -163.010,Z 1935.326,A 0.000,B 0.000,C 90.000,E1 238.742} C_DIS
LIN {X -0.045,Y -160.933,Z 1935.312,A 0.000,B 0.000,C 90.000,E1 236.135} C_DIS
LIN {X 0.066,Y -157.693,Z 1935.292,A 0.000,B 0.000,C 90.000,E1 232.557} C_DIS
LIN {X 0.004,Y -155.732,Z 1935.277,A 0.000,B 0.000,C 90.000,E1 229.908} C_DIS
LIN {X 0.057,Y -151.990,Z 1935.252,A 0.000,B 0.000,C 90.000,E1 225.405} C_DIS
LIN {X 0.073,Y -150.236,Z 1935.237,A 0.000,B 0.000,C 90.000,E1 222.690} C_DIS
LIN {X -0.004,Y -146.996,Z 1935.212,A 0.000,B 0.000,C 90.000,E1 218.177} C_DIS
LIN {X -0.014,Y -145.580,Z 1935.197,A 0.000,B 0.000,C 90.000,E1 215.438} C_DIS
